// TwinCAT 3 PLC project TcSparkplug
// Title: TcSparkplug
// Company: bstiffler582
// ProjectVersion: 0.0.1
// ProgramVersion: 3.1.4026.22
// libraries:
//   Tc2_Utilities, * (Beckhoff Automation GmbH)
//   Tc2_Standard, * (Beckhoff Automation GmbH)
//   Tc2_System, * (Beckhoff Automation GmbH)
//   Tc3_IotBase, * (Beckhoff Automation GmbH)
// project tree:
//   Util/ F_GetUnixTimestampMs.TcPOU
//   Proto/Enums/ E_ProtoWireType.TcDUT
//   Proto/ FB_ProtoReader.TcPOU, FB_ProtoWriter.TcPOU
//   Sparkplug/Enums/ E_SparkplugState.TcDUT, E_SparkplugDataType.TcDUT, E_SparkplugMessageType.TcDUT
//   Sparkplug/ F_BuildSparkplugTopic.TcPOU, FB_DDeathBuilder.TcPOU, FB_NBirthBuilder.TcPOU, FB_NDeathBuilder.TcPOU, FB_SparkplugPayload.TcPOU, FB_SparkplugDevice.TcPOU, I_SparkplugSession.TcPOU, I_SparkplugDevice.TcPOU, ST_MetricDescriptor.TcDUT, FB_SparkplugSession.TcPOU
//   Tests/ F_Assert.TcPOU, PRG_ProtoTests.TcPOU, PRG_SparkplugPayloadTests.TcPOU
// (motion and I/O tree: see PLC project test)
// real-time tasks:
//   TASK PlcTask: cycle T#10ms, priority 20, ADS port 350
//   TASK PlcTask1: cycle T#10ms, priority 21, ADS port 351

// ---- Proto/Enums/E_ProtoWireType.TcDUT
{attribute 'qualified_only'}
{attribute 'to_string'}
TYPE E_ProtoWireType :
(
	Varint          := 0,
	Fixed64         := 1,
	LengthDelimited := 2,
	Fixed32         := 5
);
END_TYPE

// ---- Sparkplug/Enums/E_SparkplugState.TcDUT
{attribute 'qualified_only'}
{attribute 'to_string'}
TYPE E_SparkplugState :
(
	Idle         := 0,	// Not started or cleanly stopped
	Connecting   := 1,	// MQTT connect in progress
	Birthing     := 2,	// NBIRTH published; waiting one cycle for device DBIRTHs
	Online       := 3,	// Fully operational
	Reconnecting := 4	// Connection lost; waiting before retry
);
END_TYPE

// ---- Sparkplug/Enums/E_SparkplugDataType.TcDUT
{attribute 'qualified_only'}
{attribute 'to_string'}
// Sparkplug B data type codes as defined in the specification.
// These are written into the `datatype` field (field 4) of every Metric.
TYPE E_SparkplugDataType :
(
	Unknown  := 0,
	Int8     := 1,
	Int16    := 2,
	Int32    := 3,
	Int64    := 4,
	UInt8    := 5,
	UInt16   := 6,
	UInt32   := 7,
	UInt64   := 8,
	Float    := 9,
	Double   := 10,
	Boolean  := 11,
	String_   := 12,
	DateTime := 13,
	Text     := 14,
	UUID     := 15,
	DataSet  := 16,
	Bytes    := 17,
	File_    := 18,   // 'File' is a reserved word in some TwinCAT versions
	Template := 19
);
END_TYPE

// ---- Sparkplug/Enums/E_SparkplugMessageType.TcDUT
{attribute 'qualified_only'}
{attribute 'to_string'}
// Sparkplug B message types.
// Note: STATE topics use a different structure (spBv1.0/STATE/{scada_host_id})
// and are handled separately in the session manager.
TYPE E_SparkplugMessageType :
(
	NBIRTH := 0,
	NDEATH := 1,
	DBIRTH := 2,
	DDEATH := 3,
	NDATA  := 4,
	DDATA  := 5,
	NCMD   := 6,
	DCMD   := 7
);
END_TYPE

// ---- Sparkplug/ST_MetricDescriptor.TcDUT
// Describes a single metric registered via FB_SparkplugDevice.AddMetric.
//
// pValue is a live pointer to the original variable in the caller's scope —
// it is dereferenced on every encode, so metric values are always current.
//
// aLastValue / sLastString hold the last-published value for change detection.
// They are updated by FB_SparkplugDevice._syncShadows() after each successful publish.
// fDeadband applies to REAL and LREAL metrics only; 0.0 means any change triggers a publish.
TYPE ST_MetricDescriptor :
STRUCT
	sName		: STRING(255);				// metric name (written in BIRTH messages)
	nAlias		: ULINT;					// alias (written in BIRTH; used alone in DATA)
	eDataType	: E_SparkplugDataType;		// Sparkplug B type code written in the metric header
	eTypeClass	: __SYSTEM.TYPE_CLASS;		// IEC type class — determines how pValue is dereferenced
	pValue		: PVOID;					// pointer to the live variable in the caller's scope
	// Change detection shadow — updated on every successful publish
	aLastValue	: ARRAY[0..7] OF BYTE;		// last-published value for non-string types (max 8 bytes)
	sLastString	: STRING(255);				// last-published value for STRING metrics
	fDeadband	: LREAL;					// minimum change to trigger a publish (REAL/LREAL only)
	bChanged	: BOOL;						// TRUE when live value differs from last-published shadow
END_STRUCT
END_TYPE

// ---- Sparkplug/I_SparkplugSession.TcPOU
// Interface consumed by device FBs to interact with the Sparkplug session.
// Decouples device FBs from the concrete FB_SparkplugSession type,
// enabling testability without a live MQTT connection.
INTERFACE I_SparkplugSession

// Returns the current seq counter and advances it (0–255 wrapping).
// Call once per outbound message to stamp the payload header.
METHOD GetNextSeq : ULINT
END_METHOD

// Returns TRUE when the session is in the Online state.
METHOD IsOnline : BOOL
END_METHOD

// Publishes a pre-encoded payload to the broker.
// Only succeeds when the session is Online or Birthing.
METHOD Publish : BOOL
VAR_INPUT
	sTopic		: STRING(255);
	pPayload	: POINTER TO BYTE;
	nLen		: UDINT;
	nQos		: UDINT;
	bRetain		: BOOL;
END_VAR
END_METHOD

// Sparkplug group ID — used by device FBs to build their own topics.
PROPERTY GroupId : STRING(127)
GET
END_GET
END_PROPERTY

// Sparkplug node ID — used by device FBs to build their own topics.
PROPERTY NodeId : STRING(127)
GET
END_GET
END_PROPERTY

END_INTERFACE

// ---- Sparkplug/I_SparkplugDevice.TcPOU
// Interface implemented by device FBs and consumed by FB_SparkplugSession
// to orchestrate the birth cycle and device lifecycle.
INTERFACE I_SparkplugDevice

// Called by the session at the start of each birth cycle, after NBIRTH is sent.
// The device must encode and publish its DBIRTH using the session's
// GetNextSeq() and Publish() methods.
METHOD OnBirth
END_METHOD

// Encodes and publishes a DDATA message using the current metric values.
// Returns FALSE if the session is not online or the publish fails.
METHOD PublishData : BOOL
VAR_INPUT
	bChangedOnly		: BOOL  := FALSE;
END_VAR
END_METHOD

// Publishes a DDEATH for this device, signalling the host that it is offline.
// Returns FALSE if the session is not online or the publish fails.
METHOD PublishDeath : BOOL
END_METHOD

// Called by the session when the device is registered via AddDevice.
// The device stores the session reference and device ID for use in OnBirth/PublishData.
METHOD SetSession
VAR_INPUT
	sDeviceId	: STRING(127);
	ipSession	: I_SparkplugSession;
END_VAR
END_METHOD

END_INTERFACE

// ---- Util/F_GetUnixTimestampMs.TcPOU
// Returns the current UTC time as milliseconds since the Unix epoch (1970-01-01 00:00:00 UTC).
// Requires: Tc2_Utilities (for F_GetSystemTime).
// F_GetSystemTime returns a ULINT of 100-nanosecond ticks since 1601-01-01 00:00:00 UTC.
FUNCTION F_GetUnixTimestampMs : ULINT

// 116444736000000000 = number of 100ns ticks from 1601-01-01 to 1970-01-01
//   = 134774 days * 86400 s/day * 10,000,000 ticks/s
// Divide by 10,000 to convert remaining 100ns ticks to milliseconds.
F_GetUnixTimestampMs := (F_GetSystemTime() - 116444736000000000) / 10000;

END_FUNCTION

// ---- Proto/FB_ProtoReader.TcPOU
FUNCTION_BLOCK FB_ProtoReader
VAR_INPUT
END_VAR
VAR_OUTPUT
END_VAR
VAR
	_pBuffer      	: POINTER TO BYTE;
	_nLength      	: UDINT;
	_nPos         	: UDINT;
	_nFieldNumber 	: UDINT;
	_eWireType    	: E_ProtoWireType;
	_bError       	: BOOL;
END_VAR

PROPERTY FieldNumber : UDINT
GET
FieldNumber := _nFieldNumber;
END_GET
END_PROPERTY

PROPERTY HasError : BOOL
GET
HasError := _bError;
END_GET
END_PROPERTY

METHOD Init
VAR_INPUT
	pBuffer 	: POINTER TO BYTE;
	nLength 	: UDINT;
END_VAR
_pBuffer      := pBuffer;
_nLength      := nLength;
_nPos         := 0;
_nFieldNumber := 0;
_bError       := FALSE;
END_METHOD

METHOD Next : BOOL
VAR_INPUT
END_VAR
VAR
	nTag : ULINT;
END_VAR
IF _bError OR _nPos >= _nLength THEN
	Next := FALSE;
	RETURN;
END_IF
IF NOT readVarintRaw(nValue => nTag) THEN
	Next := FALSE;
	RETURN;
END_IF
_nFieldNumber := ULINT_TO_UDINT(SHR(nTag, 3));
_eWireType    := ULINT_TO_INT(nTag AND 16#07);
Next := TRUE;
END_METHOD

METHOD PUBLIC ReadBool : BOOL
VAR_INPUT
END_VAR
VAR_OUTPUT
	bValue 		: BOOL;
END_VAR
VAR
	nRaw		: ULINT;
END_VAR
IF _eWireType <> E_ProtoWireType.Varint THEN _bError := TRUE; RETURN; END_IF
IF readVarintRaw(nValue => nRaw) THEN
	bValue  := nRaw <> 0;
	ReadBool := TRUE;
END_IF
END_METHOD

METHOD PUBLIC ReadBytes : BOOL
VAR_INPUT
END_VAR
VAR_OUTPUT
	pData 		: POINTER TO BYTE;
	nLen  		: UDINT;
END_VAR
VAR
	nLenRaw : ULINT;
END_VAR
IF _eWireType <> E_ProtoWireType.LengthDelimited THEN _bError := TRUE; RETURN; END_IF
IF NOT readVarintRaw(nValue => nLenRaw) THEN RETURN; END_IF
nLen := ULINT_TO_UDINT(nLenRaw);
IF _nPos + nLen > _nLength THEN _bError := TRUE; RETURN; END_IF
pData     := _pBuffer + _nPos;
_nPos     := _nPos + nLen;
ReadBytes := TRUE;
END_METHOD

METHOD PUBLIC ReadDouble : BOOL
VAR_INPUT
END_VAR
VAR_OUTPUT
	fValue 		: LREAL;
END_VAR
IF _eWireType <> E_ProtoWireType.Fixed64 OR _nPos + 8 > _nLength THEN
	_bError := TRUE; RETURN;
END_IF
MEMCPY(destAddr := ADR(fValue), srcAddr := _pBuffer + _nPos, n := 8);
_nPos      := _nPos + 8;
ReadDouble := TRUE;
END_METHOD

METHOD PUBLIC ReadFloat : BOOL
VAR_INPUT
END_VAR
VAR_OUTPUT
	fValue 		: REAL;
END_VAR
IF _eWireType <> E_ProtoWireType.Fixed32 OR _nPos + 4 > _nLength THEN
	_bError := TRUE; RETURN;
END_IF
MEMCPY(destAddr := ADR(fValue), srcAddr := _pBuffer + _nPos, n := 4);
_nPos     := _nPos + 4;
ReadFloat := TRUE;
END_METHOD

METHOD PUBLIC ReadUInt32 : BOOL
VAR_INPUT
END_VAR
VAR_OUTPUT
	nValue 		: UDINT;
END_VAR
VAR
	nRaw		: ULINT;
END_VAR
IF _eWireType <> E_ProtoWireType.Varint THEN _bError := TRUE; RETURN; END_IF
IF readVarintRaw(nValue => nRaw) THEN
	nValue    	:= ULINT_TO_UDINT(nRaw);
	ReadUInt32 	:= TRUE;
END_IF
END_METHOD

METHOD PUBLIC ReadUInt64 : BOOL
VAR_INPUT
END_VAR
VAR_OUTPUT
	nValue 		: ULINT;
END_VAR
IF _eWireType <> E_ProtoWireType.Varint THEN _bError := TRUE; RETURN; END_IF
ReadUInt64 := readVarintRaw(nValue => nValue);
END_METHOD

METHOD PRIVATE readVarintRaw : BOOL
VAR_INPUT
END_VAR
VAR_OUTPUT
	nValue 		: ULINT;
END_VAR
VAR
	nByte  		: BYTE;
	nShift 		: BYTE := 0;
END_VAR
nValue := 0;
REPEAT
	IF _nPos >= _nLength THEN
		_bError := TRUE;
		readVarintRaw := FALSE;
		RETURN;
	END_IF
	nByte  := _pBuffer[_nPos];
	_nPos  := _nPos + 1;
	nValue := nValue OR SHL(BYTE_TO_ULINT(nByte AND 16#7F), nShift);
	nShift := nShift + 7;
UNTIL (nByte AND 16#80) = 0 OR nShift >= 64
END_REPEAT;
readVarintRaw := TRUE;
END_METHOD

METHOD Skip : BOOL
VAR_INPUT
END_VAR
VAR
	nLen 		: ULINT;
END_VAR
CASE _eWireType OF
	E_ProtoWireType.Varint:
		Skip := readVarintRaw(nValue=>);  // discard
	E_ProtoWireType.Fixed32:
		IF _nPos + 4 <= _nLength THEN _nPos := _nPos + 4; Skip := TRUE; END_IF
	E_ProtoWireType.Fixed64:
		IF _nPos + 8 <= _nLength THEN _nPos := _nPos + 8; Skip := TRUE; END_IF
	E_ProtoWireType.LengthDelimited:
		IF readVarintRaw(nValue => nLen) THEN
			_nPos := _nPos + ULINT_TO_UDINT(nLen);
			Skip  := _nPos <= _nLength;
		END_IF
	ELSE
		_bError := TRUE;
END_CASE
END_METHOD

METHOD PUBLIC ReadString : BOOL
VAR_INPUT
END_VAR
VAR_OUTPUT
	sValue	: STRING(255);
END_VAR
VAR
	pData	: POINTER TO BYTE;
	nLen	: UDINT;
	nCopy	: UDINT;
	pNull	: POINTER TO BYTE;
END_VAR
IF NOT ReadBytes(pData => pData, nLen => nLen) THEN RETURN; END_IF
nCopy := MIN(nLen, 255);
MEMCPY(destAddr := ADR(sValue), srcAddr := pData, n := nCopy);
// Write null terminator at the end of the copied content
pNull  := ADR(sValue) + nCopy;
pNull^ := 0;
ReadString := TRUE;
END_METHOD

PROPERTY WireType : E_ProtoWireType
GET
WireType := _eWireType;
END_GET
END_PROPERTY

END_FUNCTION_BLOCK

// ---- Proto/FB_ProtoWriter.TcPOU
FUNCTION_BLOCK FB_ProtoWriter
VAR_INPUT
END_VAR
VAR_OUTPUT
END_VAR
VAR
	_pBuffer    	: POINTER TO BYTE;
	_nCapacity  	: UDINT;
	_nLength    	: UDINT;
	_bError     	: BOOL;
END_VAR

// Pointer to the start of the encoded bytes. Valid until the next Init call.
PROPERTY Buffer : POINTER TO BYTE
GET
Buffer := _pBuffer;
END_GET
END_PROPERTY

PROPERTY HasError : BOOL
GET
HasError := _bError;
END_GET
END_PROPERTY

METHOD Init
VAR_INPUT
	pBuffer		 		: POINTER TO BYTE;
	nCapacity			: UDINT;
END_VAR
_pBuffer   := pBuffer;
_nCapacity := nCapacity;
_nLength   := 0;
_bError    := FALSE;
END_METHOD

PROPERTY Length : UDINT
GET
Length := _nLength;
END_GET
END_PROPERTY

METHOD Reset : PVOID
VAR_INPUT
END_VAR
_nLength := 0;
_bError  := FALSE;
END_METHOD

METHOD PUBLIC WriteBool : BOOL
VAR_INPUT
	nFieldNumber 	: UDINT;
	bValue       	: BOOL;
END_VAR
WriteBool := writeTag(nFieldNumber, E_ProtoWireType.Varint)
	AND writeVarint(BOOL_TO_ULINT(bValue));
END_METHOD

METHOD PUBLIC WriteBytes : BOOL
VAR_INPUT
	nFieldNumber 	: UDINT;
	pData        	: POINTER TO BYTE;
	nLen         	: UDINT;
END_VAR
WriteBytes := writeTag(nFieldNumber, E_ProtoWireType.LengthDelimited)
	AND writeVarint(UDINT_TO_ULINT(nLen))
	AND writeRawBytes(pData, nLen);
END_METHOD

METHOD PUBLIC WriteDouble : BOOL
VAR_INPUT
	nFieldNumber 	: UDINT;
	fValue       	: LREAL;
END_VAR
VAR
	nRaw			: LWORD;
END_VAR
MEMCPY(destAddr := ADR(nRaw), srcAddr := ADR(fValue), n := 8);
WriteDouble := writeTag(nFieldNumber, E_ProtoWireType.Fixed64)
	AND writeRawBytes(ADR(nRaw), 8);
END_METHOD

METHOD PUBLIC WriteFloat : BOOL
VAR_INPUT
	nFieldNumber 	: UDINT;
	fValue       	: REAL;
END_VAR
VAR
	nRaw			: DWORD;
END_VAR
MEMCPY(destAddr := ADR(nRaw), srcAddr := ADR(fValue), n := 4);
WriteFloat := writeTag(nFieldNumber, E_ProtoWireType.Fixed32)
	AND writeRawBytes(ADR(nRaw), 4);
END_METHOD

METHOD PRIVATE writeRawByte : BOOL
VAR_INPUT
	nByte		: BYTE;
END_VAR
IF _bError OR _nLength >= _nCapacity THEN
	_bError := TRUE;
	writeRawByte := FALSE;
	RETURN;
END_IF
_pBuffer[_nLength] := nByte;
_nLength := _nLength + 1;
writeRawByte := TRUE;
END_METHOD

METHOD PRIVATE writeRawBytes : BOOL
VAR_INPUT
	pData : POINTER TO BYTE;
	nLen  : UDINT;
END_VAR
IF _bError OR (_nLength + nLen > _nCapacity) THEN
	_bError := TRUE;
	writeRawBytes := FALSE;
	RETURN;
END_IF
MEMCPY(destAddr := _pBuffer + _nLength, srcAddr := pData, n := nLen);
_nLength := _nLength + nLen;
writeRawBytes := TRUE;
END_METHOD

METHOD PUBLIC WriteString : BOOL
VAR_INPUT
	nFieldNumber 	: UDINT;
	sValue       	: STRING(255);
END_VAR
VAR
	nLen			: INT;
END_VAR
nLen := LEN(sValue);
WriteString := writeTag(nFieldNumber, E_ProtoWireType.LengthDelimited)
	AND writeVarint(TO_ULINT(nLen))
	AND writeRawBytes(ADR(sValue), TO_UDINT(nLen));
END_METHOD

METHOD PRIVATE writeTag : BOOL
VAR_INPUT
	nFieldNumber 	: UDINT;
	eWireType    	: E_ProtoWireType;
END_VAR
writeTag := writeVarint(
	SHL(UDINT_TO_ULINT(nFieldNumber), 3) OR INT_TO_ULINT(TO_INT(eWireType))
);
END_METHOD

METHOD PUBLIC WriteUInt32 : BOOL
VAR_INPUT
	nFieldNumber 	: UDINT;
	nValue       	: UDINT;
END_VAR
WriteUInt32 := writeTag(nFieldNumber, E_ProtoWireType.Varint)
	AND writeVarint(UDINT_TO_ULINT(nValue));
END_METHOD

METHOD PUBLIC WriteUInt64 : BOOL
VAR_INPUT
	nFieldNumber 	: UDINT;
  	nValue       	: ULINT;
END_VAR
WriteUInt64 := writeTag(nFieldNumber, E_ProtoWireType.Varint)
	AND writeVarint(nValue);
END_METHOD

METHOD PRIVATE writeVarint : BOOL
VAR_INPUT
	nValue		: ULINT;
END_VAR
VAR
	nByte		: BYTE;
END_VAR
IF _bError THEN writeVarint := FALSE; RETURN; END_IF
REPEAT
	nByte  := ULINT_TO_BYTE(nValue AND 16#7F);
	nValue := SHR(nValue, 7);
	IF nValue <> 0 THEN
  		nByte := nByte OR 16#80;  // more bytes follow
	END_IF
	IF NOT writeRawByte(nByte) THEN
		writeVarint := FALSE;
		RETURN;
	END_IF
UNTIL nValue = 0
END_REPEAT;
writeVarint := TRUE;
END_METHOD

END_FUNCTION_BLOCK

// ---- Sparkplug/F_BuildSparkplugTopic.TcPOU
// Builds a Sparkplug B topic string.
//
// Node-level:   spBv1.0/{group_id}/{msg_type}/{node_id}
// Device-level: spBv1.0/{group_id}/{msg_type}/{node_id}/{device_id}
//
// Pass sDeviceId := '' for node-level messages (NBIRTH, NDEATH, NDATA, NCMD).
FUNCTION F_BuildSparkplugTopic : STRING(255)
VAR_INPUT
	eMsgType	: E_SparkplugMessageType;
	sGroupId	: STRING(127);
	sNodeId		: STRING(127);
	sDeviceId	: STRING(127);
END_VAR
VAR
	sMsgType	: STRING(16);
END_VAR

CASE eMsgType OF
	E_SparkplugMessageType.NBIRTH:	sMsgType := 'NBIRTH';
	E_SparkplugMessageType.NDEATH:	sMsgType := 'NDEATH';
	E_SparkplugMessageType.DBIRTH:	sMsgType := 'DBIRTH';
	E_SparkplugMessageType.DDEATH:	sMsgType := 'DDEATH';
	E_SparkplugMessageType.NDATA:	sMsgType := 'NDATA';
	E_SparkplugMessageType.DDATA:	sMsgType := 'DDATA';
	E_SparkplugMessageType.NCMD:	sMsgType := 'NCMD';
	E_SparkplugMessageType.DCMD:	sMsgType := 'DCMD';
	ELSE							sMsgType := 'UNKNOWN';
END_CASE

F_BuildSparkplugTopic := CONCAT('spBv1.0/', sGroupId);
F_BuildSparkplugTopic := CONCAT(F_BuildSparkplugTopic, CONCAT('/', sMsgType));
F_BuildSparkplugTopic := CONCAT(F_BuildSparkplugTopic, CONCAT('/', sNodeId));

IF LEN(sDeviceId) > 0 THEN
	F_BuildSparkplugTopic := CONCAT(F_BuildSparkplugTopic, CONCAT('/', sDeviceId));
END_IF

END_FUNCTION

// ---- Sparkplug/FB_DDeathBuilder.TcPOU
// Builds a Sparkplug B DDEATH payload.
//
// DDEATH announces that a logical device is going offline. It carries only a
// timestamp and seq — no metrics. The session manager publishes it before
// disconnecting a device or on detecting a device fault.
FUNCTION_BLOCK FB_DDeathBuilder
VAR
	_aBuf		: ARRAY[0..31] OF BYTE;
	_fbPayload	: FB_SparkplugPayload;
END_VAR

// FB body intentionally empty — all logic is in Build().

METHOD Build : BOOL
VAR_INPUT
	nTimestamp	: ULINT;
	nSeq		: ULINT;
END_VAR
_fbPayload.Init(ADR(_aBuf), SIZEOF(_aBuf));
_fbPayload.WriteHeader(nTimestamp, nSeq);
Build := NOT _fbPayload.HasError;
END_METHOD

PROPERTY Payload : REFERENCE TO FB_SparkplugPayload
GET
Payload REF= _fbPayload;
END_GET
END_PROPERTY

END_FUNCTION_BLOCK

// ---- Sparkplug/FB_SparkplugPayload.TcPOU
// Incremental Sparkplug B payload builder.
//
// Wraps FB_ProtoWriter with Sparkplug-aware metric write methods. The caller
// provides an external buffer so payload capacity can be sized appropriately
// for the message type (large for NBIRTH/DBIRTH, small for DDATA).
//
// Usage:
//   fbPayload.Init(pBuffer, nCapacity);
//   fbPayload.WriteHeader(nTimestamp, nSeq);
//   fbPayload.WriteBoolMetric('MotorRunning', 1, E_SparkplugDataType.Boolean, TRUE);
//   fbPayload.WriteUInt32Metric('', 2, E_SparkplugDataType.UInt32, nSpeed);  // DATA mode: no name
//   // publish fbPayload.Buffer for fbPayload.Length bytes
//
// Metric name conventions:
//   BIRTH messages  — pass the metric name; alias is also included for future DATA messages.
//   DATA messages   — pass sName := '' to omit the name and use alias only (saves bandwidth).
//   System metrics  — pass nAlias := 0 to omit the alias field (name-only, e.g. bdSeq).
FUNCTION_BLOCK FB_SparkplugPayload
VAR
	_fbPayload		: FB_ProtoWriter;				// outer Payload message
	_fbMetric		: FB_ProtoWriter;				// inner Metric message (reused per metric)
	_aBufMetric		: ARRAY[0..511] OF BYTE;		// temp buffer for one encoded Metric
END_VAR

// FB body intentionally empty — all logic is in the methods below.

// Binds the payload builder to an external buffer and resets it.
// Must be called before any Write methods.
METHOD Init
VAR_INPUT
	pBuffer		: POINTER TO BYTE;
	nCapacity	: UDINT;
END_VAR
_fbPayload.Init(pBuffer, nCapacity);
END_METHOD

// Resets the write position without re-binding the buffer.
// Use when re-encoding into the same buffer (e.g. periodic DDATA).
METHOD Reset
_fbPayload.Reset();
END_METHOD

// Writes the Payload-level timestamp (field 1) and seq (field 4).
// Must be the first Write call after Init/Reset.
//
// Sparkplug field numbers for Payload (from sparkplug_b.proto):
//   1 = timestamp (uint64, ms since Unix epoch)
//   2 = metrics   (repeated, length-delimited)
//   3 = seq       (uint64, 0–255 wrapping)
//   4 = uuid      (string — not used by this library)
METHOD WriteHeader : BOOL
VAR_INPUT
	nTimestamp	: ULINT;
	nSeq		: ULINT;
END_VAR
WriteHeader := _fbPayload.WriteUInt64(1, nTimestamp)
	AND _fbPayload.WriteUInt64(3, nSeq);
END_METHOD

METHOD WriteBoolMetric : BOOL
VAR_INPUT
	sName		: STRING(255);
	nAlias		: ULINT;
	eDataType	: E_SparkplugDataType;
	bValue		: BOOL;
END_VAR
_fbMetric.Init(ADR(_aBufMetric), SIZEOF(_aBufMetric));
IF LEN(sName) > 0  THEN _fbMetric.WriteString(1, sName); END_IF
IF nAlias > 0      THEN _fbMetric.WriteUInt64(2, nAlias); END_IF
_fbMetric.WriteUInt32(4, TO_UDINT(eDataType));
_fbMetric.WriteBool(14, bValue);
WriteBoolMetric := _fbPayload.WriteBytes(2, ADR(_aBufMetric), _fbMetric.Length);
END_METHOD

// For Int8, Int16, Int32, UInt8, UInt16, UInt32 — encoded in proto field 10 (int_value).
METHOD WriteUInt32Metric : BOOL
VAR_INPUT
	sName		: STRING(255);
	nAlias		: ULINT;
	eDataType	: E_SparkplugDataType;
	nValue		: UDINT;
END_VAR
_fbMetric.Init(ADR(_aBufMetric), SIZEOF(_aBufMetric));
IF LEN(sName) > 0  THEN _fbMetric.WriteString(1, sName); END_IF
IF nAlias > 0      THEN _fbMetric.WriteUInt64(2, nAlias); END_IF
_fbMetric.WriteUInt32(4, TO_UDINT(eDataType));
_fbMetric.WriteUInt32(10, nValue);
WriteUInt32Metric := _fbPayload.WriteBytes(2, ADR(_aBufMetric), _fbMetric.Length);
END_METHOD

// For Int64, UInt64, DateTime — encoded in proto field 11 (long_value).
METHOD WriteUInt64Metric : BOOL
VAR_INPUT
	sName		: STRING(255);
	nAlias		: ULINT;
	eDataType	: E_SparkplugDataType;
	nValue		: ULINT;
END_VAR
_fbMetric.Init(ADR(_aBufMetric), SIZEOF(_aBufMetric));
IF LEN(sName) > 0  THEN _fbMetric.WriteString(1, sName); END_IF
IF nAlias > 0      THEN _fbMetric.WriteUInt64(2, nAlias); END_IF
_fbMetric.WriteUInt32(4, TO_UDINT(eDataType));
_fbMetric.WriteUInt64(11, nValue);
WriteUInt64Metric := _fbPayload.WriteBytes(2, ADR(_aBufMetric), _fbMetric.Length);
END_METHOD

METHOD WriteFloatMetric : BOOL
VAR_INPUT
	sName		: STRING(255);
	nAlias		: ULINT;
	eDataType	: E_SparkplugDataType;
	fValue		: REAL;
END_VAR
_fbMetric.Init(ADR(_aBufMetric), SIZEOF(_aBufMetric));
IF LEN(sName) > 0  THEN _fbMetric.WriteString(1, sName); END_IF
IF nAlias > 0      THEN _fbMetric.WriteUInt64(2, nAlias); END_IF
_fbMetric.WriteUInt32(4, TO_UDINT(eDataType));
_fbMetric.WriteFloat(12, fValue);
WriteFloatMetric := _fbPayload.WriteBytes(2, ADR(_aBufMetric), _fbMetric.Length);
END_METHOD

METHOD WriteDoubleMetric : BOOL
VAR_INPUT
	sName		: STRING(255);
	nAlias		: ULINT;
	eDataType	: E_SparkplugDataType;
	fValue		: LREAL;
END_VAR
_fbMetric.Init(ADR(_aBufMetric), SIZEOF(_aBufMetric));
IF LEN(sName) > 0  THEN _fbMetric.WriteString(1, sName); END_IF
IF nAlias > 0      THEN _fbMetric.WriteUInt64(2, nAlias); END_IF
_fbMetric.WriteUInt32(4, TO_UDINT(eDataType));
_fbMetric.WriteDouble(13, fValue);
WriteDoubleMetric := _fbPayload.WriteBytes(2, ADR(_aBufMetric), _fbMetric.Length);
END_METHOD

// For String, Text, UUID data types.
METHOD WriteStringMetric : BOOL
VAR_INPUT
	sName		: STRING(255);
	nAlias		: ULINT;
	eDataType	: E_SparkplugDataType;
	sValue		: STRING(255);
END_VAR
_fbMetric.Init(ADR(_aBufMetric), SIZEOF(_aBufMetric));
IF LEN(sName) > 0  THEN _fbMetric.WriteString(1, sName); END_IF
IF nAlias > 0      THEN _fbMetric.WriteUInt64(2, nAlias); END_IF
_fbMetric.WriteUInt32(4, TO_UDINT(eDataType));
_fbMetric.WriteString(15, sValue);
WriteStringMetric := _fbPayload.WriteBytes(2, ADR(_aBufMetric), _fbMetric.Length);
END_METHOD

// Pointer to the start of the encoded payload. Valid until the next Init call.
PROPERTY Buffer : POINTER TO BYTE
GET
Buffer := _fbPayload.Buffer;
END_GET
END_PROPERTY

PROPERTY Length : UDINT
GET
Length := _fbPayload.Length;
END_GET
END_PROPERTY

PROPERTY HasError : BOOL
GET
HasError := _fbPayload.HasError;
END_GET
END_PROPERTY

END_FUNCTION_BLOCK

// ---- Sparkplug/FB_NBirthBuilder.TcPOU
// Builds the Sparkplug B NBIRTH payload.
//
// NBIRTH announces the edge node to the Sparkplug host. It must be published
// immediately after the MQTT connection is established, before any DBIRTH or
// data messages. The seq counter is reset to 0 on every NBIRTH.
//
// This builder writes the two mandatory Sparkplug system metrics:
//   "bdSeq"                — UInt64, the birth/death sequence number.
//   "Node Control/Rebirth" — Boolean, always FALSE in the birth payload.
//                            The host writes TRUE to this metric (via NCMD)
//                            to request a full rebirth cycle.
//
// Generated code calls Payload to append node-level user metrics after Build().
//
// Usage (session manager):
//   fbNBirth.Build(nTimestamp, nBdSeq);
//   // generated node-level metrics (if any):
//   fbNBirth.Payload.WriteBoolMetric('MyNodeMetric', 1, Boolean, bValue);
//   mqttClient.Publish(sTopic, fbNBirth.Payload.Buffer, fbNBirth.Payload.Length);
FUNCTION_BLOCK FB_NBirthBuilder
VAR
	_aBuf		: ARRAY[0..2047] OF BYTE;	// 2 KB — generous for node metrics
	_fbPayload	: FB_SparkplugPayload;
END_VAR

// FB body intentionally empty — all logic is in Build().

// Initialises the payload and writes the header + system metrics.
// Call this once after connecting, before publishing NBIRTH.
// After this call, append any node-level user metrics via the Payload property.
METHOD Build : BOOL
VAR_INPUT
	nTimestamp	: ULINT;	// ms since Unix epoch
	nBdSeq		: ULINT;	// birth/death sequence number (0–255 wrapping, RETAIN)
END_VAR
_fbPayload.Init(ADR(_aBuf), SIZEOF(_aBuf));

// seq is always 0 for NBIRTH — the counter resets on every birth.
_fbPayload.WriteHeader(nTimestamp, 0);

// bdSeq: no alias — the host identifies this metric by name.
_fbPayload.WriteUInt64Metric('bdSeq', 0, E_SparkplugDataType.UInt64, nBdSeq);

// Node Control/Rebirth: no alias — identified by name.
// Value is always FALSE in the birth payload; the host sends TRUE via NCMD
// to trigger a rebirth.
_fbPayload.WriteBoolMetric('Node Control/Rebirth', 0, E_SparkplugDataType.Boolean, FALSE);

Build := NOT _fbPayload.HasError;
END_METHOD

// Exposes the underlying payload builder so generated code can append
// node-level user metrics after Build() is called.
PROPERTY Payload : REFERENCE TO FB_SparkplugPayload
GET
Payload REF= _fbPayload;
END_GET
END_PROPERTY

END_FUNCTION_BLOCK

// ---- Sparkplug/FB_NDeathBuilder.TcPOU
// Builds a Sparkplug B NDEATH payload.
//
// NDEATH is the MQTT Will message — it must be pre-built and registered with the
// broker before the MQTT connection is established. When the broker detects an
// ungraceful disconnect it publishes this payload automatically.
//
// The NDEATH payload contains exactly one metric:
//   Metric { name: "bdSeq", datatype: UInt64, long_value: <bdSeq> }
//
// No timestamp and no seq field are included per the Sparkplug B specification.
//
// Usage:
//   fbNDeath.Build(nBdSeq);
//   mqttClient.SetWill(
//     sTopic  := F_BuildSparkplugTopic(NDEATH, sGroup, sNode, ''),
//     pPayload := fbNDeath.PayloadBuffer,
//     nLen     := fbNDeath.PayloadLength);
FUNCTION_BLOCK FB_NDeathBuilder
VAR
	// Internal buffers — owned by this FB, stable between Build() calls.
	_aBufMetric		: ARRAY[0..31] OF BYTE;
	_aBufPayload	: ARRAY[0..47] OF BYTE;

	_fbMetric		: FB_ProtoWriter;
	_fbPayload		: FB_ProtoWriter;

	_nPayloadLength	: UDINT;
	_bValid			: BOOL;
END_VAR

// FB body intentionally empty — all logic is in Build().

// Encodes the NDEATH payload for the given birth/death sequence number.
// Call this once before registering the MQTT Will, and again after each
// reconnect if the bdSeq value has changed.
METHOD Build : BOOL
VAR_INPUT
	nBdSeq	: ULINT;
END_VAR
// ── Encode the bdSeq metric ──────────────────────────────────────────────────
// Sparkplug field numbers for Metric:
//   1 = name (string)
//   4 = datatype (uint32)
//  11 = long_value (uint64) — used for UInt64 and Int64 values
_fbMetric.Init(ADR(_aBufMetric), SIZEOF(_aBufMetric));
_fbMetric.WriteString(1,  'bdSeq');
_fbMetric.WriteUInt32(4,  TO_UDINT(E_SparkplugDataType.UInt64));
_fbMetric.WriteUInt64(11, nBdSeq);

// ── Encode the Payload ────────────────────────────────────────────────────────
// Sparkplug field numbers for Payload:
//   2 = metrics (repeated, length-delimited)
// Intentionally omitting timestamp (f1) and seq (f4) — not required in NDEATH.
_fbPayload.Init(ADR(_aBufPayload), SIZEOF(_aBufPayload));
_fbPayload.WriteBytes(2, ADR(_aBufMetric), _fbMetric.Length);

_bValid         := NOT _fbMetric.HasError AND NOT _fbPayload.HasError;
_nPayloadLength := _fbPayload.Length;
Build           := _bValid;
END_METHOD

// TRUE if the last Build() call succeeded without buffer overflow.
PROPERTY IsValid : BOOL
GET
IsValid := _bValid;
END_GET
END_PROPERTY

// Pointer to the encoded payload bytes. Valid until the next Build() call.
PROPERTY PayloadBuffer : POINTER TO BYTE
GET
PayloadBuffer := ADR(_aBufPayload);
END_GET
END_PROPERTY

// Number of encoded bytes. Zero if Build() has not been called yet.
PROPERTY PayloadLength : UDINT
GET
PayloadLength := _nPayloadLength;
END_GET
END_PROPERTY

END_FUNCTION_BLOCK

// ---- Sparkplug/FB_SparkplugDevice.TcPOU
// Generic Sparkplug B device function block.
//
// Register metrics once at startup via AddMetric(), then pass this FB to the
// session via AddDevice(). The session will call OnBirth() automatically on
// every birth cycle; the caller decides when to send DDATA by calling PublishData().
//
// Usage:
//   fbDevice.AddMetric('Speed',       1, nMotorSpeed);
//   fbDevice.AddMetric('Running',     2, bMotorRunning);
//   fbDevice.AddMetric('Temperature', 3, fMotorTemp);
//   fbSpkSession.AddDevice('Motor1', fbDevice);
//   // ...
//   IF tPublish.Q THEN fbDevice.PublishData(); END_IF
//
// AddMetric() stores a live pointer to the caller's variable — do not call it
// more than once per metric, and ensure the variable outlives this FB.
//
// Call this FB every PLC cycle. It runs change detection and sets bDataPending
// when at least one metric's live value differs from its last-published shadow.
// The caller then decides when to call PublishData() (e.g. on bDataPending rising edge).
FUNCTION_BLOCK FB_SparkplugDevice IMPLEMENTS I_SparkplugDevice
VAR_INPUT
	// Default deadband applied to all REAL and LREAL metrics at AddMetric time.
	// Per-metric overrides are available via SetDeadband(). 0.0 = any change triggers a publish.
	fDefaultDeadband	: LREAL := 0.0;
	// When TRUE the FB publishes DDATA automatically on any detected change.
	// The caller may still call PublishData() independently (e.g. periodic refresh).
	bAutoPublish		: BOOL  := FALSE;
END_VAR
VAR_OUTPUT
	// TRUE when at least one metric's live value differs from its last-published shadow.
	// Recomputed every cycle — if a value changes and reverts before PublishData() is called,
	// this returns FALSE (correct report-by-exception behaviour).
	bDataPending		: BOOL;
END_VAR
VAR
	_aMetrics		: ARRAY[0..15] OF ST_MetricDescriptor;
	_nMetricCount	: UDINT;

	_sDeviceId		: STRING(127);
	_ipSession		: I_SparkplugSession;

	_sBirthTopic	: STRING(255);
	_sDataTopic		: STRING(255);
	_sDeathTopic	: STRING(255);

	_aBirthBuf		: ARRAY[0..2047] OF BYTE;
	_aDataBuf		: ARRAY[0..511] OF BYTE;
	_fbBirthPayload	: FB_SparkplugPayload;
	_fbDataPayload	: FB_SparkplugPayload;
	_fbDeath		: FB_DDeathBuilder;
END_VAR

// Run change detection every cycle once a session is attached.
IF _ipSession <> 0 THEN
	_checkChanges();
	IF bAutoPublish AND bDataPending THEN
		PublishData(bChangedOnly := TRUE);
	END_IF
END_IF

// Encodes all registered metrics into fbPayload.
// bBirthMode = TRUE  → writes name + alias (DBIRTH).
// bBirthMode = FALSE → writes alias only (DDATA — saves bandwidth).
METHOD PRIVATE _writeMetrics
VAR_IN_OUT
	fbPayload	: FB_SparkplugPayload;
END_VAR
VAR_INPUT
	bBirthMode		: BOOL;
	bChangedOnly	: BOOL := FALSE;	// when TRUE, skips metrics whose bChanged flag is FALSE
END_VAR
VAR
	i		: UDINT;
	sName	: STRING(255);
	pBool	: POINTER TO BOOL;
	pSint	: POINTER TO SINT;
	pInt	: POINTER TO INT;
	pDint	: POINTER TO DINT;
	pLint	: POINTER TO LINT;
	pUsint	: POINTER TO USINT;
	pUint	: POINTER TO UINT;
	pUdint	: POINTER TO UDINT;
	pUlint	: POINTER TO ULINT;
	pByte	: POINTER TO BYTE;
	pWord	: POINTER TO WORD;
	pDword	: POINTER TO DWORD;
	pLword	: POINTER TO LWORD;
	pReal	: POINTER TO REAL;
	pLreal	: POINTER TO LREAL;
	pStr	: POINTER TO STRING(255);
END_VAR
IF _nMetricCount = 0 THEN RETURN; END_IF

FOR i := 0 TO _nMetricCount - 1 DO
	// In changed-only mode skip metrics that haven't changed since last publish.
	IF bChangedOnly AND NOT _aMetrics[i].bChanged THEN
		;
	ELSE
	// In BIRTH mode write the metric name; in DATA mode write alias only.
	sName := SEL(bBirthMode, '', _aMetrics[i].sName);

	CASE _aMetrics[i].eTypeClass OF
		__SYSTEM.TYPE_CLASS.TYPE_BOOL:
			pBool  := _aMetrics[i].pValue;
			fbPayload.WriteBoolMetric(sName, _aMetrics[i].nAlias, _aMetrics[i].eDataType, pBool^);

		__SYSTEM.TYPE_CLASS.TYPE_SINT:
			pSint  := _aMetrics[i].pValue;
			fbPayload.WriteUInt32Metric(sName, _aMetrics[i].nAlias, _aMetrics[i].eDataType, TO_UDINT(pSint^));

		__SYSTEM.TYPE_CLASS.TYPE_INT:
			pInt   := _aMetrics[i].pValue;
			fbPayload.WriteUInt32Metric(sName, _aMetrics[i].nAlias, _aMetrics[i].eDataType, TO_UDINT(pInt^));

		__SYSTEM.TYPE_CLASS.TYPE_DINT:
			pDint  := _aMetrics[i].pValue;
			fbPayload.WriteUInt32Metric(sName, _aMetrics[i].nAlias, _aMetrics[i].eDataType, TO_UDINT(pDint^));

		__SYSTEM.TYPE_CLASS.TYPE_LINT:
			pLint  := _aMetrics[i].pValue;
			fbPayload.WriteUInt64Metric(sName, _aMetrics[i].nAlias, _aMetrics[i].eDataType, TO_ULINT(pLint^));

		__SYSTEM.TYPE_CLASS.TYPE_USINT:
			pUsint := _aMetrics[i].pValue;
			fbPayload.WriteUInt32Metric(sName, _aMetrics[i].nAlias, _aMetrics[i].eDataType, TO_UDINT(pUsint^));

		__SYSTEM.TYPE_CLASS.TYPE_UINT:
			pUint  := _aMetrics[i].pValue;
			fbPayload.WriteUInt32Metric(sName, _aMetrics[i].nAlias, _aMetrics[i].eDataType, TO_UDINT(pUint^));

		__SYSTEM.TYPE_CLASS.TYPE_UDINT:
			pUdint := _aMetrics[i].pValue;
			fbPayload.WriteUInt32Metric(sName, _aMetrics[i].nAlias, _aMetrics[i].eDataType, pUdint^);

		__SYSTEM.TYPE_CLASS.TYPE_ULINT:
			pUlint := _aMetrics[i].pValue;
			fbPayload.WriteUInt64Metric(sName, _aMetrics[i].nAlias, _aMetrics[i].eDataType, pUlint^);

		__SYSTEM.TYPE_CLASS.TYPE_BYTE:
			pByte  := _aMetrics[i].pValue;
			fbPayload.WriteUInt32Metric(sName, _aMetrics[i].nAlias, _aMetrics[i].eDataType, TO_UDINT(pByte^));

		__SYSTEM.TYPE_CLASS.TYPE_WORD:
			pWord  := _aMetrics[i].pValue;
			fbPayload.WriteUInt32Metric(sName, _aMetrics[i].nAlias, _aMetrics[i].eDataType, TO_UDINT(pWord^));

		__SYSTEM.TYPE_CLASS.TYPE_DWORD:
			pDword := _aMetrics[i].pValue;
			fbPayload.WriteUInt32Metric(sName, _aMetrics[i].nAlias, _aMetrics[i].eDataType, TO_UDINT(pDword^));

		__SYSTEM.TYPE_CLASS.TYPE_LWORD:
			pLword := _aMetrics[i].pValue;
			fbPayload.WriteUInt64Metric(sName, _aMetrics[i].nAlias, _aMetrics[i].eDataType, TO_ULINT(pLword^));

		__SYSTEM.TYPE_CLASS.TYPE_REAL:
			pReal  := _aMetrics[i].pValue;
			fbPayload.WriteFloatMetric(sName, _aMetrics[i].nAlias, _aMetrics[i].eDataType, pReal^);

		__SYSTEM.TYPE_CLASS.TYPE_LREAL:
			pLreal := _aMetrics[i].pValue;
			fbPayload.WriteDoubleMetric(sName, _aMetrics[i].nAlias, _aMetrics[i].eDataType, pLreal^);

		__SYSTEM.TYPE_CLASS.TYPE_STRING:
			pStr   := _aMetrics[i].pValue;
			fbPayload.WriteStringMetric(sName, _aMetrics[i].nAlias, _aMetrics[i].eDataType, pStr^);
	END_CASE
	END_IF
END_FOR
END_METHOD

// Registers a metric to be included in DBIRTH and DDATA messages.
// Infers the Sparkplug B data type from the IEC type of value.
// Call once per metric during startup before AddDevice().
//
// Supported types: BOOL, SINT/INT/DINT/LINT, USINT/UINT/UDINT/ULINT,
//                  BYTE/WORD/DWORD/LWORD, REAL, LREAL, STRING(n)
METHOD AddMetric
VAR_INPUT
	sName	: STRING(255);
	nAlias	: ULINT;
	value	: ANY;
END_VAR
VAR
	eDataType	: E_SparkplugDataType;
END_VAR
IF _nMetricCount >= 16 THEN RETURN; END_IF

// Map IEC TypeClass → Sparkplug B data type code
CASE value.TypeClass OF
	__SYSTEM.TYPE_CLASS.TYPE_BOOL	: eDataType := E_SparkplugDataType.Boolean;
	__SYSTEM.TYPE_CLASS.TYPE_SINT	: eDataType := E_SparkplugDataType.Int8;
	__SYSTEM.TYPE_CLASS.TYPE_INT	: eDataType := E_SparkplugDataType.Int16;
	__SYSTEM.TYPE_CLASS.TYPE_DINT	: eDataType := E_SparkplugDataType.Int32;
	__SYSTEM.TYPE_CLASS.TYPE_LINT	: eDataType := E_SparkplugDataType.Int64;
	__SYSTEM.TYPE_CLASS.TYPE_USINT	: eDataType := E_SparkplugDataType.UInt8;
	__SYSTEM.TYPE_CLASS.TYPE_UINT	: eDataType := E_SparkplugDataType.UInt16;
	__SYSTEM.TYPE_CLASS.TYPE_UDINT	: eDataType := E_SparkplugDataType.UInt32;
	__SYSTEM.TYPE_CLASS.TYPE_ULINT	: eDataType := E_SparkplugDataType.UInt64;
	__SYSTEM.TYPE_CLASS.TYPE_BYTE	: eDataType := E_SparkplugDataType.UInt8;
	__SYSTEM.TYPE_CLASS.TYPE_WORD	: eDataType := E_SparkplugDataType.UInt16;
	__SYSTEM.TYPE_CLASS.TYPE_DWORD	: eDataType := E_SparkplugDataType.UInt32;
	__SYSTEM.TYPE_CLASS.TYPE_LWORD	: eDataType := E_SparkplugDataType.UInt64;
	__SYSTEM.TYPE_CLASS.TYPE_REAL	: eDataType := E_SparkplugDataType.Float;
	__SYSTEM.TYPE_CLASS.TYPE_LREAL	: eDataType := E_SparkplugDataType.Double;
	__SYSTEM.TYPE_CLASS.TYPE_STRING	: eDataType := E_SparkplugDataType.String_;
ELSE
	eDataType := E_SparkplugDataType.Unknown;
END_CASE

_aMetrics[_nMetricCount].sName		 := sName;
_aMetrics[_nMetricCount].nAlias		 := nAlias;
_aMetrics[_nMetricCount].eDataType	 := eDataType;
_aMetrics[_nMetricCount].eTypeClass  := value.TypeClass;
_aMetrics[_nMetricCount].pValue		 := value.pValue;

// Apply default deadband to float types; all others use exact-match comparison.
_aMetrics[_nMetricCount].fDeadband := 0.0;
IF value.TypeClass = __SYSTEM.TYPE_CLASS.TYPE_REAL
OR value.TypeClass = __SYSTEM.TYPE_CLASS.TYPE_LREAL THEN
	_aMetrics[_nMetricCount].fDeadband := fDefaultDeadband;
END_IF

_nMetricCount := _nMetricCount + 1;
END_METHOD

// Called by the session on each birth cycle after NBIRTH is published.
// Builds topics, encodes the DBIRTH payload, and publishes it.
METHOD OnBirth
// Build topics — GroupId and NodeId are valid once the session has been called at least once.
_sBirthTopic := F_BuildSparkplugTopic(E_SparkplugMessageType.DBIRTH, _ipSession.GroupId, _ipSession.NodeId, _sDeviceId);
_sDataTopic  := F_BuildSparkplugTopic(E_SparkplugMessageType.DDATA,  _ipSession.GroupId, _ipSession.NodeId, _sDeviceId);
_sDeathTopic := F_BuildSparkplugTopic(E_SparkplugMessageType.DDEATH, _ipSession.GroupId, _ipSession.NodeId, _sDeviceId);

_fbBirthPayload.Init(ADR(_aBirthBuf), SIZEOF(_aBirthBuf));
_fbBirthPayload.WriteHeader(F_GetUnixTimestampMs(), _ipSession.GetNextSeq());
_writeMetrics(_fbBirthPayload, TRUE);
_ipSession.Publish(_sBirthTopic, _fbBirthPayload.Buffer, _fbBirthPayload.Length, 1, FALSE);

// Sync shadows after birth so change detection starts from the just-published values.
_syncShadows();
END_METHOD

// Encodes and publishes a DDATA message.
// bChangedOnly = FALSE (default): sends all metrics — use for periodic refreshes.
// bChangedOnly = TRUE: sends only metrics whose value has changed since the last publish.
// Returns FALSE if the session is not online or the publish fails.
METHOD PublishData : BOOL
VAR_INPUT
	bChangedOnly	: BOOL := FALSE;
END_VAR
IF NOT _ipSession.IsOnline() THEN RETURN; END_IF

_fbDataPayload.Init(ADR(_aDataBuf), SIZEOF(_aDataBuf));
_fbDataPayload.WriteHeader(F_GetUnixTimestampMs(), _ipSession.GetNextSeq());
_writeMetrics(_fbDataPayload, FALSE, bChangedOnly);
PublishData := _ipSession.Publish(_sDataTopic, _fbDataPayload.Buffer, _fbDataPayload.Length, 1, FALSE);

// Sync only the shadows that were written so bChanged stays accurate for any skipped metrics.
IF PublishData THEN
	_syncShadows(bChangedOnly);
END_IF
END_METHOD

// Publishes a DDEATH for this device, signalling the host that it is offline.
// Returns FALSE if the session is not online or the publish fails.
METHOD PublishDeath : BOOL
IF NOT _ipSession.IsOnline() THEN RETURN; END_IF

_fbDeath.Build(F_GetUnixTimestampMs(), _ipSession.GetNextSeq());
PublishDeath := _ipSession.Publish(_sDeathTopic, _fbDeath.Payload.Buffer, _fbDeath.Payload.Length, 1, FALSE);
END_METHOD

// Called by FB_SparkplugSession.AddDevice — stores the device ID and session reference.
// Do not call directly.
METHOD SetSession
VAR_INPUT
	sDeviceId	: STRING(127);
	ipSession	: I_SparkplugSession;
END_VAR
_sDeviceId := sDeviceId;
_ipSession := ipSession;
END_METHOD

// Recomputes bDataPending by comparing each metric's live value against its last-published shadow.
// Floats use deadband comparison; all other types use byte-exact MEMCMP.
// The shadow is NOT updated here — only _syncShadows() writes to it.
METHOD PRIVATE _checkChanges
VAR
	i			: UDINT;
	nSize		: UDINT;
	pStr		: POINTER TO STRING(255);
	pReal		: POINTER TO REAL;
	pLastReal	: POINTER TO REAL;
	pLreal		: POINTER TO LREAL;
	pLastLreal	: POINTER TO LREAL;
END_VAR
bDataPending := FALSE;

FOR i := 0 TO _nMetricCount - 1 DO
	_aMetrics[i].bChanged := FALSE;

	CASE _aMetrics[i].eTypeClass OF
		__SYSTEM.TYPE_CLASS.TYPE_STRING:
			pStr := _aMetrics[i].pValue;
			IF pStr^ <> _aMetrics[i].sLastString THEN
				_aMetrics[i].bChanged := TRUE;
			END_IF

		__SYSTEM.TYPE_CLASS.TYPE_REAL:
			pReal		:= _aMetrics[i].pValue;
			pLastReal	:= ADR(_aMetrics[i].aLastValue);
			IF ABS(pReal^ - pLastReal^) > TO_REAL(_aMetrics[i].fDeadband) THEN
				_aMetrics[i].bChanged := TRUE;
			END_IF

		__SYSTEM.TYPE_CLASS.TYPE_LREAL:
			pLreal		:= _aMetrics[i].pValue;
			pLastLreal	:= ADR(_aMetrics[i].aLastValue);
			IF ABS(pLreal^ - pLastLreal^) > _aMetrics[i].fDeadband THEN
				_aMetrics[i].bChanged := TRUE;
			END_IF
	ELSE
		nSize := _typeSize(_aMetrics[i].eTypeClass);
		IF nSize > 0 AND MEMCMP(_aMetrics[i].pValue, ADR(_aMetrics[i].aLastValue), nSize) <> 0 THEN
			_aMetrics[i].bChanged := TRUE;
		END_IF
	END_CASE

	bDataPending := bDataPending OR _aMetrics[i].bChanged;
END_FOR
END_METHOD

// Returns the byte width of the given IEC type class.
// Returns 0 for STRING (handled separately) and unknown types.
METHOD PRIVATE _typeSize : UDINT
VAR_INPUT
	eTypeClass	: __SYSTEM.TYPE_CLASS;
END_VAR
CASE eTypeClass OF
	__SYSTEM.TYPE_CLASS.TYPE_BOOL,
	__SYSTEM.TYPE_CLASS.TYPE_SINT,
	__SYSTEM.TYPE_CLASS.TYPE_USINT,
	__SYSTEM.TYPE_CLASS.TYPE_BYTE	: _typeSize := 1;
	__SYSTEM.TYPE_CLASS.TYPE_INT,
	__SYSTEM.TYPE_CLASS.TYPE_UINT,
	__SYSTEM.TYPE_CLASS.TYPE_WORD	: _typeSize := 2;
	__SYSTEM.TYPE_CLASS.TYPE_DINT,
	__SYSTEM.TYPE_CLASS.TYPE_UDINT,
	__SYSTEM.TYPE_CLASS.TYPE_DWORD,
	__SYSTEM.TYPE_CLASS.TYPE_REAL	: _typeSize := 4;
	__SYSTEM.TYPE_CLASS.TYPE_LINT,
	__SYSTEM.TYPE_CLASS.TYPE_ULINT,
	__SYSTEM.TYPE_CLASS.TYPE_LWORD,
	__SYSTEM.TYPE_CLASS.TYPE_LREAL	: _typeSize := 8;
ELSE
	_typeSize := 0; // STRING or unknown — handled separately
END_CASE
END_METHOD

// Copies the current live value of every metric into its shadow (last-published record).
// Called after a confirmed DBIRTH or DDATA publish.
METHOD PRIVATE _syncShadows
VAR_INPUT
	bChangedOnly	: BOOL := FALSE;	// when TRUE, only syncs metrics whose bChanged flag is TRUE
END_VAR
VAR
	i		: UDINT;
	nSize	: UDINT;
	pStr	: POINTER TO STRING(255);
END_VAR
FOR i := 0 TO _nMetricCount - 1 DO
	IF bChangedOnly AND NOT _aMetrics[i].bChanged THEN
		;
	ELSIF _aMetrics[i].eTypeClass = __SYSTEM.TYPE_CLASS.TYPE_STRING THEN
		pStr := _aMetrics[i].pValue;
		_aMetrics[i].sLastString := pStr^;
	ELSE
		nSize := _typeSize(_aMetrics[i].eTypeClass);
		IF nSize > 0 THEN
			MEMCPY(ADR(_aMetrics[i].aLastValue), _aMetrics[i].pValue, nSize);
		END_IF
	END_IF
END_FOR
END_METHOD

// Overrides the deadband for a single REAL or LREAL metric identified by its alias.
// Call after AddMetric() and before the first birth cycle.
// Has no effect on non-float metrics (their comparison is always byte-exact).
METHOD SetDeadband
VAR_INPUT
	nAlias		: ULINT;
	fDeadband	: LREAL;
END_VAR
VAR
	i	: UDINT;
END_VAR
FOR i := 0 TO _nMetricCount - 1 DO
	IF _aMetrics[i].nAlias = nAlias THEN
		_aMetrics[i].fDeadband := fDeadband;
		RETURN;
	END_IF
END_FOR
END_METHOD

END_FUNCTION_BLOCK

// ---- Sparkplug/FB_SparkplugSession.TcPOU
// Sparkplug B session manager.
//
// Manages the full Sparkplug lifecycle: MQTT connection, Will registration,
// NBIRTH/NDEATH sequencing, rebirth on command, and reconnection with backoff.
//
// Caller responsibilities:
//   - Declare nBdSeq as RETAIN so it survives power cycles.
//   - Call this FB every PLC cycle regardless of state.
//   - When bBirthRequired rises, publish DBIRTH for every device in the same cycle.
//   - Use GetNextSeq() and Publish() for all outbound data messages.
//
// NOTE: The MQTT client calls (Connect, Subscribe, Publish) target the
// Beckhoff TF6701 Tc3_IotBase FB_IotMqttClient API. Verify method signatures
// against your installed TF6701 version if compile errors occur.

// TODO: support for TLS, certs...
// maybe pass in refrence to MqttClient?
FUNCTION_BLOCK FB_SparkplugSession IMPLEMENTS I_SparkplugSession
VAR_INPUT
	sGroupId		: STRING(127);
	sNodeId			: STRING(127);
	fbMqttClient	: REFERENCE TO FB_IotMqttClient;
	bEnable			: BOOL;
END_VAR
VAR_OUTPUT
	eState			: E_SparkplugState;
	bOnline			: BOOL;
	bBirthRequired	: BOOL;				// TRUE for one cycle — publish DBIRTH on this cycle
	bError			: BOOL;
	sErrorMsg		: STRING(255);
END_VAR
VAR_IN_OUT
	// IMPORTANT: declare this variable as RETAIN in the calling program.
	// It must survive power cycles to satisfy the Sparkplug B specification.
	nBdSeq			: ULINT;
END_VAR
VAR
	_fbNDeath		: FB_NDeathBuilder;
	_fbNBirth		: FB_NBirthBuilder;

	_nSeq			: ULINT;			// 0–255 wrapping; reset to 0 on NBIRTH, 1 after
	_bConnect		: BOOL;

	// Cached topic strings (built once on enable)
	_sNbirthTopic	: STRING(255);
	_sNdeathTopic	: STRING(255);
	_sNcmdTopic		: STRING(255);

	// MQTT Will — must remain stable in memory while the connection is live
	_stWill			: ST_IotMqttWill;

	// Reconnect backoff
	_tReconnect		: TON;

	// One-shot flags
	_bLastEnable		: BOOL;
	_bBirthSignalled	: BOOL;		// TRUE after bBirthRequired was set high this birth cycle
	_bRebirthPending	: BOOL;		// Set by NCMD handler; causes Online→Birthing transition
	_bWasOnline			: BOOL;		// TRUE if connection dropped from Online or Birthing

	// Inbound message processing
	_fbMsg			: FB_IotMqttMessage;
	_fbMsgQueue 	: FB_IotMqttMessageQueue;
	_sMsgTopic		: STRING(255);
	_fbReader		: FB_ProtoReader;
	_fbInnerReader	: FB_ProtoReader;
	_pMetricData	: POINTER TO BYTE;
	_nMetricLen		: UDINT;
	_sMetricName	: STRING(255);
	_bMetricBool	: BOOL;

	// Registered devices — called on each birth cycle
	_aDevices		: ARRAY[0..15] OF I_SparkplugDevice;
	_nDeviceCount	: UDINT;
	_iDev			: UDINT;
END_VAR

fbMqttClient.Execute(_bConnect);

bOnline := (eState = E_SparkplugState.Online);
bError  := fbMqttClient.bError;

// ── State machine ─────────────────────────────────────────────────────────────
CASE eState OF

// ─────────────────────────────────────────────────────────────────────────────
E_SparkplugState.Idle:
	bBirthRequired  := FALSE;
	_bBirthSignalled := FALSE;
	_bWasOnline      := FALSE;

	IF bEnable AND NOT _bLastEnable THEN
		_sNbirthTopic := F_BuildSparkplugTopic(E_SparkplugMessageType.NBIRTH, sGroupId, sNodeId, '');
		_sNdeathTopic := F_BuildSparkplugTopic(E_SparkplugMessageType.NDEATH, sGroupId, sNodeId, '');
		_sNcmdTopic   := F_BuildSparkplugTopic(E_SparkplugMessageType.NCMD,   sGroupId, sNodeId, '');
		sErrorMsg     := '';
		beginConnect();
		eState := E_SparkplugState.Connecting;
	END_IF

// ─────────────────────────────────────────────────────────────────────────────
E_SparkplugState.Connecting:
	IF NOT bEnable THEN
		_bConnect := FALSE;
		eState := E_SparkplugState.Idle;

	ELSIF fbMqttClient.bError THEN
		sErrorMsg := 'Connect failed';
		// bdSeq does NOT increment here — the Will was never registered with a broker
		_tReconnect(IN := FALSE);
		eState := E_SparkplugState.Reconnecting;

	ELSIF fbMqttClient.bConnected THEN
		fbMqttClient.ipMessageQueue := _fbMsgQueue;
		fbMqttClient.Subscribe(_sNcmdTopic, 1);
		eState := E_SparkplugState.Birthing;
	END_IF

// ─────────────────────────────────────────────────────────────────────────────
E_SparkplugState.Birthing:
	IF NOT bEnable OR fbMqttClient.bError OR NOT fbMqttClient.bConnected THEN
		// Connection dropped while birthing — Will has been registered so bdSeq must advance
		nBdSeq := (nBdSeq + 1) MOD 256;
		_bBirthSignalled := FALSE;
		_tReconnect(IN := FALSE);
		IF NOT bEnable THEN
			_bCOnnect := FALSE;
			eState := E_SparkplugState.Idle;
		ELSE
			sErrorMsg := 'Connection lost during birth';
			eState    := E_SparkplugState.Reconnecting;
		END_IF

	ELSIF NOT _bBirthSignalled THEN
		// First half of birth cycle: publish NBIRTH and raise the birth flag
		_nSeq := 0;
		_fbNBirth.Build(F_GetUnixTimestampMs(), nBdSeq);
		fbMqttClient.Publish(
			sTopic       := _sNbirthTopic,
			pPayload     := _fbNBirth.Payload.Buffer,
			nPayloadSize := _fbNBirth.Payload.Length,
			eQos         := TcIotMqttQos.AtLeastOnceDelivery,
			bRetain      := FALSE);
		_nSeq := 1;		// First DBIRTH will use seq=1

		// Publish DBIRTH for every registered device (seq=1, 2, ...)
		IF _nDeviceCount > 0 THEN
			FOR _iDev := 0 TO _nDeviceCount - 1 DO
				IF _aDevices[_iDev] <> 0 THEN
					_aDevices[_iDev].OnBirth();
				END_IF
			END_FOR
		END_IF

		bBirthRequired   := TRUE;	// Signal any external device FBs for one cycle
		_bBirthSignalled := TRUE;

	ELSE
		// Second half: device FBs have had one cycle to see bBirthRequired — go Online
		bBirthRequired   := FALSE;
		_bBirthSignalled := FALSE;
		_bWasOnline      := TRUE;
		eState           := E_SparkplugState.Online;
	END_IF

// ─────────────────────────────────────────────────────────────────────────────
E_SparkplugState.Online:
	IF NOT bEnable THEN
		_bConnect := FALSE;
		nBdSeq := (nBdSeq + 1) MOD 256;
		eState := E_SparkplugState.Idle;

	ELSIF fbMqttClient.bError OR NOT fbMqttClient.bConnected THEN
		sErrorMsg := 'Connection lost';
		nBdSeq    := (nBdSeq + 1) MOD 256;
		_tReconnect(IN := FALSE);
		eState := E_SparkplugState.Reconnecting;

	ELSIF _bRebirthPending THEN
		// Soft rebirth (triggered by NCMD or STATE recovery) — bdSeq does NOT change
		_bRebirthPending := FALSE;
		_bBirthSignalled := FALSE;
		eState           := E_SparkplugState.Birthing;

	ELSE
		pollMessages();
	END_IF

// ─────────────────────────────────────────────────────────────────────────────
E_SparkplugState.Reconnecting:
	_tReconnect(IN := TRUE, PT := T#5S);

	IF NOT bEnable THEN
		_tReconnect(IN := FALSE);
		eState := E_SparkplugState.Idle;

	ELSIF _tReconnect.Q THEN
		_tReconnect(IN := FALSE);
		beginConnect();
		eState := E_SparkplugState.Connecting;
	END_IF

END_CASE

_bLastEnable := bEnable;

// Registers a device FB with the session.
// The session will call ipDevice.OnBirth() automatically on every birth cycle.
// Call once during startup after AddMetric(), before the first birth cycle.
METHOD AddDevice
VAR_INPUT
	sDeviceId	: STRING(127);
	ipDevice	: I_SparkplugDevice;
END_VAR
VAR
	ipMe	: I_SparkplugSession;
END_VAR
IF _nDeviceCount >= 16 THEN RETURN; END_IF

ipMe := THIS^;
ipDevice.SetSession(sDeviceId, ipMe);
_aDevices[_nDeviceCount] := ipDevice;
_nDeviceCount := _nDeviceCount + 1;
END_METHOD

// Builds the NDEATH Will payload from the current nBdSeq, then initiates
// the MQTT connection. nBdSeq must already be at the correct value for this
// connection before this method is called.
METHOD PRIVATE beginConnect
// Build NDEATH — this becomes the MQTT Will payload.
// The broker will publish it automatically on ungraceful disconnect.
_fbNDeath.Build(nBdSeq);

_stWill.sTopic			:= _sNdeathTopic;
_stWill.pPayload     	:= _fbNDeath.PayloadBuffer;
_stWill.nPayloadSize 	:= _fbNDeath.PayloadLength;
_stWill.eQos         	:= TcIotMqttQos.AtLeastOnceDelivery;
_stWill.bRetain      	:= FALSE;

fbMqttClient.stWill 		:= _stWill;

_bConnect := TRUE;
END_METHOD

// Returns the current seq value and advances the counter (0–255 wrapping).
// Device FBs must call this once per published message to stamp the payload header.
METHOD GetNextSeq : ULINT
GetNextSeq := _nSeq;
_nSeq      := (_nSeq + 1) MOD 256;
END_METHOD

// Returns the Sparkplug group ID configured on this session.
// Device FBs use this to build their own topics without duplicating the group/node at the call site.
PROPERTY GroupId : STRING(127)
GET
GroupId := sGroupId;
END_GET
END_PROPERTY

// Parses an NCMD payload. Sets _bRebirthPending if Node Control/Rebirth = TRUE.
// All other node commands are ignored here; device DCMDs are handled by device FBs.
METHOD PRIVATE handleNcmd
VAR_INPUT
	pPayload	: PVOID;
	nLen		: UDINT;
END_VAR
VAR
	pMetric		: POINTER TO BYTE;
	nMetricLen	: UDINT;
	sName		: STRING(255);
	bBoolVal	: BOOL;
	bGotName	: BOOL;
	bGotBool	: BOOL;
END_VAR
// Decode the outer Payload message — we only care about Metric entries (field 2)
_fbReader.Init(pPayload, nLen);
WHILE _fbReader.Next() DO
	IF _fbReader.FieldNumber = 2 THEN
		_fbReader.ReadBytes(pData => pMetric, nLen => nMetricLen);

		// Decode the inner Metric message
		sName    := '';
		bBoolVal := FALSE;
		bGotName := FALSE;
		bGotBool := FALSE;

		_fbInnerReader.Init(pMetric, nMetricLen);
		WHILE _fbInnerReader.Next() DO
			CASE _fbInnerReader.FieldNumber OF
				1:	// name
					_fbInnerReader.ReadString(sValue => sName);
					bGotName := TRUE;
				14:	// boolean_value
					_fbInnerReader.ReadBool(bValue => bBoolVal);
					bGotBool := TRUE;
			ELSE
				_fbInnerReader.Skip();
			END_CASE
		END_WHILE

		IF bGotName AND bGotBool
			AND sName = 'Node Control/Rebirth'
			AND bBoolVal
		THEN
			_bRebirthPending := TRUE;
		END_IF
	ELSE
		_fbReader.Skip();
	END_IF
END_WHILE
END_METHOD

// Returns TRUE when the session is in the Online state.
// Implements I_SparkplugSession — avoids naming conflict with the bOnline VAR_OUTPUT.
METHOD IsOnline : BOOL
IsOnline := bOnline;
END_METHOD

// Returns the Sparkplug node ID configured on this session.
// Device FBs use this to build their own topics without duplicating the group/node at the call site.
PROPERTY NodeId : STRING(127)
GET
NodeId := sNodeId;
END_GET
END_PROPERTY

// Drains the inbound message queue for this cycle.
// Dispatches NCMD messages to handleNcmd; all other topics are silently discarded.
METHOD PRIVATE pollMessages
// Drain one message per cycle.
// The Sparkplug B spec requires the primary application to send NCMD/rebirth
// to edge nodes after it reconnects, so rebirth is driven by NCMD only.
IF _fbMsgQueue.nQueuedMessages > 0 AND _fbMsgQueue.Dequeue(_fbMsg) THEN
	_fbMsg.GetTopic(ADR(_sMsgTopic), 255);
	IF _sMsgTopic = _sNcmdTopic THEN
		handleNcmd(_fbMsg.pPayload, _fbMsg.nPayloadSize);
	END_IF
END_IF
END_METHOD

// Publishes a pre-encoded payload. Device FBs use this to send DBIRTH and DDATA.
// Only call when bOnline is TRUE or bBirthRequired is TRUE.
METHOD Publish : BOOL
VAR_INPUT
	sTopic		: STRING(255);
	pPayload	: POINTER TO BYTE;
	nLen		: UDINT;
	nQos		: UDINT := 1;
	bRetain		: BOOL  := FALSE;
END_VAR
IF eState = E_SparkplugState.Online OR eState = E_SparkplugState.Birthing THEN
	Publish := fbMqttClient.Publish(
		sTopic       := sTopic,
		pPayload     := pPayload,
		nPayloadSize := nLen,
		eQos         := UDINT_TO_SINT(nQos),
		bRetain      := bRetain);
END_IF
END_METHOD

END_FUNCTION_BLOCK

// ---- Tests/F_Assert.TcPOU
// Increments nPass if bCondition is TRUE, otherwise increments nFail and records
// the name of the first failure in sFirstFail.
FUNCTION F_Assert : BOOL
VAR_INPUT
	bCondition	: BOOL;
	sTestName	: STRING(255);
END_VAR
VAR_IN_OUT
	nPass		: UDINT;
	nFail		: UDINT;
	sFirstFail	: STRING(255);
END_VAR

IF bCondition THEN
	nPass    := nPass + 1;
	F_Assert := TRUE;
ELSE
	nFail := nFail + 1;
	IF nFail = 1 THEN
		sFirstFail := sTestName;
	END_IF
	F_Assert := FALSE;
END_IF

END_FUNCTION

// ---- Tests/PRG_ProtoTests.TcPOU
// Proto round-trip test suite.
// Set bRun := TRUE to execute. Results appear in nPass, nFail, bAllPassed, sFirstFail.
PROGRAM PRG_ProtoTests
VAR
	// Trigger
	bRun		: BOOL;
	_bLastRun	: BOOL;

	// Results
	nPass		: UDINT;
	nFail		: UDINT;
	bAllPassed	: BOOL;
	sFirstFail	: STRING(255);
	bRan		: BOOL;

	// Shared writer / reader
	fbW			: FB_ProtoWriter;
	fbR			: FB_ProtoReader;

	// Second writer for nested-message test
	fbWInner	: FB_ProtoWriter;

	// Buffers
	aBuf		: ARRAY[0..511] OF BYTE;
	aBufInner	: ARRAY[0..63]  OF BYTE;
	aSmallBuf	: ARRAY[0..3]   OF BYTE;   // intentionally tiny for overflow test

	// Known byte sequence used in the Bytes test
	aTestBytes	: ARRAY[0..3] OF BYTE := [16#DE, 16#AD, 16#BE, 16#EF];

	// Readback variables
	nU32		: UDINT;
	nU64		: ULINT;
	bVal		: BOOL;
	fVal		: REAL;
	dVal		: LREAL;
	sVal		: STRING(255);
	pBytes		: POINTER TO BYTE;
	nBytesLen	: UDINT;
END_VAR

// Run once per rising edge of bRun
IF NOT (bRun AND NOT _bLastRun) THEN
	_bLastRun := bRun;
	RETURN;
END_IF
_bLastRun := bRun;

nPass      := 0;
nFail      := 0;
sFirstFail := '';
bRan       := FALSE;

// ── T01: UInt32 — single-byte varint (value fits in 7 bits) ──────────────────
fbW.Init(ADR(aBuf), SIZEOF(aBuf));
fbW.WriteUInt32(1, 5);
fbR.Init(ADR(aBuf), fbW.Length);
fbR.Next();
fbR.ReadUInt32(nValue => nU32);
F_Assert(
	bCondition := fbR.FieldNumber = 1 AND nU32 = 5 AND NOT fbR.HasError,
	sTestName  := 'T01 UInt32 single-byte varint',
	nPass := nPass, nFail := nFail, sFirstFail := sFirstFail);

// ── T02: UInt32 — multi-byte varint (value > 127, needs 2 bytes) ─────────────
fbW.Init(ADR(aBuf), SIZEOF(aBuf));
fbW.WriteUInt32(2, 300);
fbR.Init(ADR(aBuf), fbW.Length);
fbR.Next();
fbR.ReadUInt32(nValue => nU32);
F_Assert(
	bCondition := fbR.FieldNumber = 2 AND nU32 = 300 AND NOT fbR.HasError,
	sTestName  := 'T02 UInt32 multi-byte varint',
	nPass := nPass, nFail := nFail, sFirstFail := sFirstFail);

// ── T03: UInt64 — Sparkplug-realistic timestamp (10-byte varint) ─────────────
fbW.Init(ADR(aBuf), SIZEOF(aBuf));
fbW.WriteUInt64(3, 1700000000000);
fbR.Init(ADR(aBuf), fbW.Length);
fbR.Next();
fbR.ReadUInt64(nValue => nU64);
F_Assert(
	bCondition := fbR.FieldNumber = 3 AND nU64 = 1700000000000 AND NOT fbR.HasError,
	sTestName  := 'T03 UInt64 large value',
	nPass := nPass, nFail := nFail, sFirstFail := sFirstFail);

// ── T04: Bool TRUE ────────────────────────────────────────────────────────────
fbW.Init(ADR(aBuf), SIZEOF(aBuf));
fbW.WriteBool(4, TRUE);
fbR.Init(ADR(aBuf), fbW.Length);
fbR.Next();
fbR.ReadBool(bValue => bVal);
F_Assert(
	bCondition := fbR.FieldNumber = 4 AND bVal = TRUE AND NOT fbR.HasError,
	sTestName  := 'T04 Bool TRUE',
	nPass := nPass, nFail := nFail, sFirstFail := sFirstFail);

// ── T05: Bool FALSE ───────────────────────────────────────────────────────────
fbW.Init(ADR(aBuf), SIZEOF(aBuf));
fbW.WriteBool(5, FALSE);
fbR.Init(ADR(aBuf), fbW.Length);
fbR.Next();
fbR.ReadBool(bValue => bVal);
F_Assert(
	bCondition := fbR.FieldNumber = 5 AND bVal = FALSE AND NOT fbR.HasError,
	sTestName  := 'T05 Bool FALSE',
	nPass := nPass, nFail := nFail, sFirstFail := sFirstFail);

// ── T06: Float (Fixed32 wire type) ───────────────────────────────────────────
// 1.5 is exactly representable in IEEE 754 — safe for exact equality check.
fbW.Init(ADR(aBuf), SIZEOF(aBuf));
fbW.WriteFloat(6, 1.5);
fbR.Init(ADR(aBuf), fbW.Length);
fbR.Next();
fbR.ReadFloat(fValue => fVal);
F_Assert(
	bCondition := fbR.FieldNumber = 6 AND fVal = 1.5 AND NOT fbR.HasError,
	sTestName  := 'T06 Float round-trip',
	nPass := nPass, nFail := nFail, sFirstFail := sFirstFail);

// ── T07: Double (Fixed64 wire type) ──────────────────────────────────────────
// 0.125 = 2^-3, exactly representable.
fbW.Init(ADR(aBuf), SIZEOF(aBuf));
fbW.WriteDouble(7, 0.125);
fbR.Init(ADR(aBuf), fbW.Length);
fbR.Next();
fbR.ReadDouble(fValue => dVal);
F_Assert(
	bCondition := fbR.FieldNumber = 7 AND dVal = 0.125 AND NOT fbR.HasError,
	sTestName  := 'T07 Double round-trip',
	nPass := nPass, nFail := nFail, sFirstFail := sFirstFail);

// ── T08: String ───────────────────────────────────────────────────────────────
fbW.Init(ADR(aBuf), SIZEOF(aBuf));
fbW.WriteString(8, 'hello');
fbR.Init(ADR(aBuf), fbW.Length);
fbR.Next();
fbR.ReadString(sValue => sVal);
F_Assert(
	bCondition := fbR.FieldNumber = 8 AND sVal = 'hello' AND NOT fbR.HasError,
	sTestName  := 'T08 String round-trip',
	nPass := nPass, nFail := nFail, sFirstFail := sFirstFail);

// ── T09: Bytes ────────────────────────────────────────────────────────────────
fbW.Init(ADR(aBuf), SIZEOF(aBuf));
fbW.WriteBytes(9, ADR(aTestBytes), SIZEOF(aTestBytes));
fbR.Init(ADR(aBuf), fbW.Length);
fbR.Next();
fbR.ReadBytes(pData => pBytes, nLen => nBytesLen);
F_Assert(
	bCondition := fbR.FieldNumber = 9
		AND nBytesLen = 4
		AND pBytes[0] = 16#DE AND pBytes[1] = 16#AD
		AND pBytes[2] = 16#BE AND pBytes[3] = 16#EF
		AND NOT fbR.HasError,
	sTestName  := 'T09 Bytes round-trip',
	nPass := nPass, nFail := nFail, sFirstFail := sFirstFail);

// ── T10: Multiple fields written and read in sequence ─────────────────────────
fbW.Init(ADR(aBuf), SIZEOF(aBuf));
fbW.WriteUInt32(1, 42);
fbW.WriteBool(2, TRUE);
fbW.WriteFloat(3, 1.5);
fbR.Init(ADR(aBuf), fbW.Length);

fbR.Next(); fbR.ReadUInt32(nValue => nU32);
F_Assert(
	bCondition := fbR.FieldNumber = 1 AND nU32 = 42,
	sTestName  := 'T10a Multi-field field 1',
	nPass := nPass, nFail := nFail, sFirstFail := sFirstFail);

fbR.Next(); fbR.ReadBool(bValue => bVal);
F_Assert(
	bCondition := fbR.FieldNumber = 2 AND bVal = TRUE,
	sTestName  := 'T10b Multi-field field 2',
	nPass := nPass, nFail := nFail, sFirstFail := sFirstFail);

fbR.Next(); fbR.ReadFloat(fValue => fVal);
F_Assert(
	bCondition := fbR.FieldNumber = 3 AND fVal = 1.5,
	sTestName  := 'T10c Multi-field field 3',
	nPass := nPass, nFail := nFail, sFirstFail := sFirstFail);

F_Assert(
	bCondition := NOT fbR.Next(),
	sTestName  := 'T10d Multi-field end of buffer',
	nPass := nPass, nFail := nFail, sFirstFail := sFirstFail);

// ── T11: Skip ────────────────────────────────────────────────────────────────
// Write fields 1 and 3; skip field 1 and verify field 3 is read correctly.
fbW.Init(ADR(aBuf), SIZEOF(aBuf));
fbW.WriteUInt32(1, 99);
fbW.WriteFloat(2, 2.5);    // Fixed32 — exercises Skip for that wire type too
fbW.WriteUInt32(3, 77);
fbR.Init(ADR(aBuf), fbW.Length);

fbR.Next(); fbR.Skip();   // skip UInt32
fbR.Next(); fbR.Skip();   // skip Float
fbR.Next(); fbR.ReadUInt32(nValue => nU32);
F_Assert(
	bCondition := fbR.FieldNumber = 3 AND nU32 = 77 AND NOT fbR.HasError,
	sTestName  := 'T11 Skip fields',
	nPass := nPass, nFail := nFail, sFirstFail := sFirstFail);

// ── T12: Nested message — minimal Sparkplug Metric inside a Payload ───────────
// Inner: Metric { alias=1 (f2), datatype=11/Boolean (f4), boolean_value=true (f14) }
fbWInner.Init(ADR(aBufInner), SIZEOF(aBufInner));
fbWInner.WriteUInt64(2,  1);    // alias
fbWInner.WriteUInt32(4, 11);    // datatype = Boolean
fbWInner.WriteBool(14, TRUE);   // boolean_value

// Outer: Payload { timestamp (f1), metrics (f2) }
fbW.Init(ADR(aBuf), SIZEOF(aBuf));
fbW.WriteUInt64(1, 1700000000000);
fbW.WriteBytes(2, ADR(aBufInner), fbWInner.Length);

// Decode outer payload
fbR.Init(ADR(aBuf), fbW.Length);
fbR.Next(); fbR.ReadUInt64(nValue => nU64);
F_Assert(
	bCondition := fbR.FieldNumber = 1 AND nU64 = 1700000000000,
	sTestName  := 'T12a Nested outer timestamp',
	nPass := nPass, nFail := nFail, sFirstFail := sFirstFail);

fbR.Next(); fbR.ReadBytes(pData => pBytes, nLen => nBytesLen);
F_Assert(
	bCondition := fbR.FieldNumber = 2 AND nBytesLen = fbWInner.Length AND NOT fbR.HasError,
	sTestName  := 'T12b Nested metrics field',
	nPass := nPass, nFail := nFail, sFirstFail := sFirstFail);

// Re-use fbR to decode the inner metric bytes (zero-copy — pBytes points into aBuf)
fbR.Init(pBytes, nBytesLen);

fbR.Next(); fbR.ReadUInt64(nValue => nU64);
F_Assert(
	bCondition := fbR.FieldNumber = 2 AND nU64 = 1,
	sTestName  := 'T12c Nested metric alias',
	nPass := nPass, nFail := nFail, sFirstFail := sFirstFail);

fbR.Next(); fbR.ReadUInt32(nValue => nU32);
F_Assert(
	bCondition := fbR.FieldNumber = 4 AND nU32 = 11,
	sTestName  := 'T12d Nested metric datatype',
	nPass := nPass, nFail := nFail, sFirstFail := sFirstFail);

fbR.Next(); fbR.ReadBool(bValue => bVal);
F_Assert(
	bCondition := fbR.FieldNumber = 14 AND bVal = TRUE AND NOT fbR.HasError,
	sTestName  := 'T12e Nested metric boolean_value',
	nPass := nPass, nFail := nFail, sFirstFail := sFirstFail);

// ── T13: Writer overflow ──────────────────────────────────────────────────────
// aSmallBuf is 4 bytes; a UInt64 field for 1700000000000 encodes to 11 bytes.
fbW.Init(ADR(aSmallBuf), SIZEOF(aSmallBuf));
fbW.WriteUInt64(1, 1700000000000);
F_Assert(
	bCondition := fbW.HasError,
	sTestName  := 'T13 Writer overflow sets HasError',
	nPass := nPass, nFail := nFail, sFirstFail := sFirstFail);

// ── T14: Reader wire type mismatch ───────────────────────────────────────────
// Field is encoded as Fixed32 (Float); reading it as Varint (UInt32) must error.
fbW.Init(ADR(aBuf), SIZEOF(aBuf));
fbW.WriteFloat(1, 1.5);
fbR.Init(ADR(aBuf), fbW.Length);
fbR.Next();
fbR.ReadUInt32(nValue => nU32);   // wrong read type
F_Assert(
	bCondition := fbR.HasError,
	sTestName  := 'T14 Reader wire type mismatch sets HasError',
	nPass := nPass, nFail := nFail, sFirstFail := sFirstFail);

// ── Done ─────────────────────────────────────────────────────────────────────
bAllPassed := (nFail = 0);
bRan       := TRUE;

END_PROGRAM

// ---- Tests/PRG_SparkplugPayloadTests.TcPOU
// Sparkplug payload builder test suite.
// Set bRun := TRUE to execute. Results in nPass, nFail, bAllPassed, sFirstFail.
PROGRAM PRG_SparkplugPayloadTests
VAR
	bRun		: BOOL;
	_bLastRun	: BOOL;

	nPass		: UDINT;
	nFail		: UDINT;
	bAllPassed	: BOOL;
	sFirstFail	: STRING(255);
	bRan		: BOOL;

	// Builders under test
	fbNDeath	: FB_NDeathBuilder;
	fbNBirth	: FB_NBirthBuilder;
	fbDDeath	: FB_DDeathBuilder;

	// Generic payload builder for metric writer tests
	aBuf		: ARRAY[0..511] OF BYTE;
	fbPayload	: FB_SparkplugPayload;

	// Readers
	fbR			: FB_ProtoReader;
	fbRInner	: FB_ProtoReader;

	// Readback vars
	nU32		: UDINT;
	nU64		: ULINT;
	bVal		: BOOL;
	fVal		: REAL;
	dVal		: LREAL;
	sVal		: STRING(255);
	pMetric		: POINTER TO BYTE;
	nMetricLen	: UDINT;

	// Fixed test values
	nTestTs		: ULINT := 1700000000000;	// ms — a Sparkplug-realistic timestamp
	nTestBdSeq	: ULINT := 42;
	nTestSeq	: ULINT := 7;
END_VAR

IF NOT (bRun AND NOT _bLastRun) THEN
	_bLastRun := bRun;
	RETURN;
END_IF
_bLastRun := bRun;

nPass      := 0;
nFail      := 0;
sFirstFail := '';
bRan       := FALSE;

// ════════════════════════════════════════════════════════════════════════════
// GROUP 1 — F_BuildSparkplugTopic
// ════════════════════════════════════════════════════════════════════════════

// T01: Node-level topic — no device ID
F_Assert(
	bCondition := F_BuildSparkplugTopic(E_SparkplugMessageType.NBIRTH, 'Grp', 'Node', '') = 'spBv1.0/Grp/NBIRTH/Node',
	sTestName  := 'T01 Topic node-level NBIRTH',
	nPass := nPass, nFail := nFail, sFirstFail := sFirstFail);

// T02: Device-level topic — device ID appended
F_Assert(
	bCondition := F_BuildSparkplugTopic(E_SparkplugMessageType.DDATA, 'G', 'N', 'D') = 'spBv1.0/G/DDATA/N/D',
	sTestName  := 'T02 Topic device-level DDATA',
	nPass := nPass, nFail := nFail, sFirstFail := sFirstFail);

// T03: NCMD node-level
F_Assert(
	bCondition := F_BuildSparkplugTopic(E_SparkplugMessageType.NCMD, 'Plant1', 'PLC1', '') = 'spBv1.0/Plant1/NCMD/PLC1',
	sTestName  := 'T03 Topic NCMD',
	nPass := nPass, nFail := nFail, sFirstFail := sFirstFail);

// T04: NDEATH
F_Assert(
	bCondition := F_BuildSparkplugTopic(E_SparkplugMessageType.NDEATH, 'Grp', 'Node', '') = 'spBv1.0/Grp/NDEATH/Node',
	sTestName  := 'T04 Topic NDEATH',
	nPass := nPass, nFail := nFail, sFirstFail := sFirstFail);


// ════════════════════════════════════════════════════════════════════════════
// GROUP 2 — FB_NDeathBuilder
// Expected outer payload: f2 (metric) only — no timestamp, no seq.
// Expected inner metric:  f1=name, f4=datatype, f11=long_value
// ════════════════════════════════════════════════════════════════════════════

fbNDeath.Build(nTestBdSeq);
fbR.Init(fbNDeath.PayloadBuffer, fbNDeath.PayloadLength);

// T05: builder reports no error
F_Assert(
	bCondition := fbNDeath.IsValid,
	sTestName  := 'T05 NDeathBuilder IsValid',
	nPass := nPass, nFail := nFail, sFirstFail := sFirstFail);

// T06: first (and only) outer field is the metrics field (f2) — no timestamp or seq
fbR.Next();
F_Assert(
	bCondition := fbR.FieldNumber = 2,
	sTestName  := 'T06 NDEATH outer field is metrics (f2), no header fields',
	nPass := nPass, nFail := nFail, sFirstFail := sFirstFail);

// T07–T10: decode the inner bdSeq metric
fbR.ReadBytes(pData => pMetric, nLen => nMetricLen);
fbRInner.Init(pMetric, nMetricLen);

fbRInner.Next(); fbRInner.ReadString(sValue => sVal);
F_Assert(
	bCondition := fbRInner.FieldNumber = 1 AND sVal = 'bdSeq',
	sTestName  := 'T07 NDEATH metric name = bdSeq',
	nPass := nPass, nFail := nFail, sFirstFail := sFirstFail);

fbRInner.Next(); fbRInner.ReadUInt32(nValue => nU32);
F_Assert(
	bCondition := fbRInner.FieldNumber = 4 AND nU32 = TO_UDINT(E_SparkplugDataType.UInt64),
	sTestName  := 'T08 NDEATH metric datatype = UInt64',
	nPass := nPass, nFail := nFail, sFirstFail := sFirstFail);

fbRInner.Next(); fbRInner.ReadUInt64(nValue => nU64);
F_Assert(
	bCondition := fbRInner.FieldNumber = 11 AND nU64 = nTestBdSeq,
	sTestName  := 'T09 NDEATH metric long_value = bdSeq',
	nPass := nPass, nFail := nFail, sFirstFail := sFirstFail);

F_Assert(
	bCondition := NOT fbRInner.Next() AND NOT fbR.Next(),
	sTestName  := 'T10 NDEATH no extra fields in metric or payload',
	nPass := nPass, nFail := nFail, sFirstFail := sFirstFail);


// ════════════════════════════════════════════════════════════════════════════
// GROUP 3 — FB_NBirthBuilder
// Expected outer payload: f1=timestamp, f3=seq(0), f2=bdSeq metric, f2=Rebirth metric
// bdSeq metric inner:    f1=name, f4=datatype, f11=long_value  (no alias: alias=0)
// Rebirth metric inner:  f1=name, f4=datatype, f14=boolean_value
// ════════════════════════════════════════════════════════════════════════════

fbNBirth.Build(nTestTs, nTestBdSeq);
fbR.Init(fbNBirth.Payload.Buffer, fbNBirth.Payload.Length);

// T11: builder reports no error
F_Assert(
	bCondition := NOT fbNBirth.Payload.HasError,
	sTestName  := 'T11 NBirthBuilder no error',
	nPass := nPass, nFail := nFail, sFirstFail := sFirstFail);

// T12–T13: outer header
fbR.Next(); fbR.ReadUInt64(nValue => nU64);
F_Assert(
	bCondition := fbR.FieldNumber = 1 AND nU64 = nTestTs,
	sTestName  := 'T12 NBIRTH timestamp correct',
	nPass := nPass, nFail := nFail, sFirstFail := sFirstFail);

fbR.Next(); fbR.ReadUInt64(nValue => nU64);
F_Assert(
	bCondition := fbR.FieldNumber = 3 AND nU64 = 0,
	sTestName  := 'T13 NBIRTH seq = 0',
	nPass := nPass, nFail := nFail, sFirstFail := sFirstFail);

// T14–T16: first metric — bdSeq
fbR.Next(); fbR.ReadBytes(pData => pMetric, nLen => nMetricLen);
F_Assert(
	bCondition := fbR.FieldNumber = 2,
	sTestName  := 'T14 NBIRTH first metric field present',
	nPass := nPass, nFail := nFail, sFirstFail := sFirstFail);

fbRInner.Init(pMetric, nMetricLen);
fbRInner.Next(); fbRInner.ReadString(sValue => sVal);
F_Assert(
	bCondition := fbRInner.FieldNumber = 1 AND sVal = 'bdSeq',
	sTestName  := 'T15 NBIRTH bdSeq metric name',
	nPass := nPass, nFail := nFail, sFirstFail := sFirstFail);

fbRInner.Next(); fbRInner.ReadUInt32(nValue => nU32);
fbRInner.Next(); fbRInner.ReadUInt64(nValue => nU64);
F_Assert(
	bCondition := nU32 = TO_UDINT(E_SparkplugDataType.UInt64) AND nU64 = nTestBdSeq,
	sTestName  := 'T16 NBIRTH bdSeq metric datatype and value',
	nPass := nPass, nFail := nFail, sFirstFail := sFirstFail);

// T17–T19: second metric — Node Control/Rebirth
fbR.Next(); fbR.ReadBytes(pData => pMetric, nLen => nMetricLen);
F_Assert(
	bCondition := fbR.FieldNumber = 2,
	sTestName  := 'T17 NBIRTH second metric field present',
	nPass := nPass, nFail := nFail, sFirstFail := sFirstFail);

fbRInner.Init(pMetric, nMetricLen);
fbRInner.Next(); fbRInner.ReadString(sValue => sVal);
F_Assert(
	bCondition := fbRInner.FieldNumber = 1 AND sVal = 'Node Control/Rebirth',
	sTestName  := 'T18 NBIRTH Rebirth metric name',
	nPass := nPass, nFail := nFail, sFirstFail := sFirstFail);

fbRInner.Next(); fbRInner.ReadUInt32(nValue => nU32);
fbRInner.Next(); fbRInner.ReadBool(bValue => bVal);
F_Assert(
	bCondition := nU32 = TO_UDINT(E_SparkplugDataType.Boolean) AND bVal = FALSE,
	sTestName  := 'T19 NBIRTH Rebirth metric datatype and value=FALSE',
	nPass := nPass, nFail := nFail, sFirstFail := sFirstFail);

F_Assert(
	bCondition := NOT fbR.Next(),
	sTestName  := 'T20 NBIRTH no extra outer fields',
	nPass := nPass, nFail := nFail, sFirstFail := sFirstFail);


// ════════════════════════════════════════════════════════════════════════════
// GROUP 4 — FB_DDeathBuilder
// Expected outer payload: f1=timestamp, f3=seq — no metrics follow.
// ════════════════════════════════════════════════════════════════════════════

fbDDeath.Build(nTestTs, nTestSeq);
fbR.Init(fbDDeath.Payload.Buffer, fbDDeath.Payload.Length);

fbR.Next(); fbR.ReadUInt64(nValue => nU64);
F_Assert(
	bCondition := fbR.FieldNumber = 1 AND nU64 = nTestTs,
	sTestName  := 'T21 DDEATH timestamp correct',
	nPass := nPass, nFail := nFail, sFirstFail := sFirstFail);

fbR.Next(); fbR.ReadUInt64(nValue => nU64);
F_Assert(
	bCondition := fbR.FieldNumber = 3 AND nU64 = nTestSeq,
	sTestName  := 'T22 DDEATH seq correct',
	nPass := nPass, nFail := nFail, sFirstFail := sFirstFail);

F_Assert(
	bCondition := NOT fbR.Next(),
	sTestName  := 'T23 DDEATH no metrics',
	nPass := nPass, nFail := nFail, sFirstFail := sFirstFail);


// ════════════════════════════════════════════════════════════════════════════
// GROUP 5 — FB_SparkplugPayload metric writers
// Helper pattern for each test:
//   Init → WriteHeader → WriteXxxMetric → decode outer (skip f1+f4) → decode inner
// ════════════════════════════════════════════════════════════════════════════

// ── T24–T27: WriteBoolMetric — birth mode (name + alias + datatype + value) ─
fbPayload.Init(ADR(aBuf), SIZEOF(aBuf));
fbPayload.WriteHeader(nTestTs, 0);
fbPayload.WriteBoolMetric('Running', 1, E_SparkplugDataType.Boolean, TRUE);

fbR.Init(fbPayload.Buffer, fbPayload.Length);
fbR.Next(); fbR.Skip();		// f1: timestamp
fbR.Next(); fbR.Skip();		// f3: seq
fbR.Next(); fbR.ReadBytes(pData => pMetric, nLen => nMetricLen);

fbRInner.Init(pMetric, nMetricLen);
fbRInner.Next(); fbRInner.ReadString(sValue => sVal);
F_Assert(
	bCondition := fbRInner.FieldNumber = 1 AND sVal = 'Running',
	sTestName  := 'T24 WriteBoolMetric name',
	nPass := nPass, nFail := nFail, sFirstFail := sFirstFail);

fbRInner.Next(); fbRInner.ReadUInt64(nValue => nU64);
F_Assert(
	bCondition := fbRInner.FieldNumber = 2 AND nU64 = 1,
	sTestName  := 'T25 WriteBoolMetric alias',
	nPass := nPass, nFail := nFail, sFirstFail := sFirstFail);

fbRInner.Next(); fbRInner.ReadUInt32(nValue => nU32);
F_Assert(
	bCondition := fbRInner.FieldNumber = 4 AND nU32 = TO_UDINT(E_SparkplugDataType.Boolean),
	sTestName  := 'T26 WriteBoolMetric datatype',
	nPass := nPass, nFail := nFail, sFirstFail := sFirstFail);

fbRInner.Next(); fbRInner.ReadBool(bValue => bVal);
F_Assert(
	bCondition := fbRInner.FieldNumber = 14 AND bVal = TRUE,
	sTestName  := 'T27 WriteBoolMetric value',
	nPass := nPass, nFail := nFail, sFirstFail := sFirstFail);

// ── T28–T29: WriteBoolMetric — data mode (no name; first field must be alias) ─
fbPayload.Init(ADR(aBuf), SIZEOF(aBuf));
fbPayload.WriteHeader(nTestTs, 5);
fbPayload.WriteBoolMetric('', 3, E_SparkplugDataType.Boolean, FALSE);

fbR.Init(fbPayload.Buffer, fbPayload.Length);
fbR.Next(); fbR.Skip();
fbR.Next(); fbR.Skip();
fbR.Next(); fbR.ReadBytes(pData => pMetric, nLen => nMetricLen);

fbRInner.Init(pMetric, nMetricLen);
fbRInner.Next();
F_Assert(
	bCondition := fbRInner.FieldNumber = 2,
	sTestName  := 'T28 WriteBoolMetric data mode: first field is alias (no name)',
	nPass := nPass, nFail := nFail, sFirstFail := sFirstFail);
fbRInner.ReadUInt64(nValue => nU64);
F_Assert(
	bCondition := nU64 = 3,
	sTestName  := 'T29 WriteBoolMetric data mode: alias value correct',
	nPass := nPass, nFail := nFail, sFirstFail := sFirstFail);

// ── T30–T31: WriteUInt32Metric (int_value → proto field 10) ─────────────────
fbPayload.Init(ADR(aBuf), SIZEOF(aBuf));
fbPayload.WriteHeader(nTestTs, 0);
fbPayload.WriteUInt32Metric('Speed', 2, E_SparkplugDataType.UInt32, 1500);

fbR.Init(fbPayload.Buffer, fbPayload.Length);
fbR.Next(); fbR.Skip(); fbR.Next(); fbR.Skip();
fbR.Next(); fbR.ReadBytes(pData => pMetric, nLen => nMetricLen);

fbRInner.Init(pMetric, nMetricLen);
fbRInner.Next(); fbRInner.Skip();		// f1: name
fbRInner.Next(); fbRInner.Skip();		// f2: alias
fbRInner.Next(); fbRInner.ReadUInt32(nValue => nU32);
F_Assert(
	bCondition := fbRInner.FieldNumber = 4 AND nU32 = TO_UDINT(E_SparkplugDataType.UInt32),
	sTestName  := 'T30 WriteUInt32Metric datatype',
	nPass := nPass, nFail := nFail, sFirstFail := sFirstFail);

fbRInner.Next(); fbRInner.ReadUInt32(nValue => nU32);
F_Assert(
	bCondition := fbRInner.FieldNumber = 10 AND nU32 = 1500,
	sTestName  := 'T31 WriteUInt32Metric int_value (f10)',
	nPass := nPass, nFail := nFail, sFirstFail := sFirstFail);

// ── T32–T33: WriteFloatMetric (float_value → proto field 12) ────────────────
fbPayload.Init(ADR(aBuf), SIZEOF(aBuf));
fbPayload.WriteHeader(nTestTs, 0);
fbPayload.WriteFloatMetric('Temp', 3, E_SparkplugDataType.Float, 2.5);

fbR.Init(fbPayload.Buffer, fbPayload.Length);
fbR.Next(); fbR.Skip(); fbR.Next(); fbR.Skip();
fbR.Next(); fbR.ReadBytes(pData => pMetric, nLen => nMetricLen);

fbRInner.Init(pMetric, nMetricLen);
fbRInner.Next(); fbRInner.Skip();		// f1: name
fbRInner.Next(); fbRInner.Skip();		// f2: alias
fbRInner.Next(); fbRInner.ReadUInt32(nValue => nU32);
F_Assert(
	bCondition := fbRInner.FieldNumber = 4 AND nU32 = TO_UDINT(E_SparkplugDataType.Float),
	sTestName  := 'T32 WriteFloatMetric datatype',
	nPass := nPass, nFail := nFail, sFirstFail := sFirstFail);

fbRInner.Next(); fbRInner.ReadFloat(fValue => fVal);
F_Assert(
	bCondition := fbRInner.FieldNumber = 12 AND fVal = 2.5,
	sTestName  := 'T33 WriteFloatMetric float_value (f12)',
	nPass := nPass, nFail := nFail, sFirstFail := sFirstFail);

// ── T34–T35: WriteDoubleMetric (double_value → proto field 13) ──────────────
fbPayload.Init(ADR(aBuf), SIZEOF(aBuf));
fbPayload.WriteHeader(nTestTs, 0);
fbPayload.WriteDoubleMetric('Pressure', 4, E_SparkplugDataType.Double, 0.125);

fbR.Init(fbPayload.Buffer, fbPayload.Length);
fbR.Next(); fbR.Skip(); fbR.Next(); fbR.Skip();
fbR.Next(); fbR.ReadBytes(pData => pMetric, nLen => nMetricLen);

fbRInner.Init(pMetric, nMetricLen);
fbRInner.Next(); fbRInner.Skip();
fbRInner.Next(); fbRInner.Skip();
fbRInner.Next(); fbRInner.ReadUInt32(nValue => nU32);
F_Assert(
	bCondition := fbRInner.FieldNumber = 4 AND nU32 = TO_UDINT(E_SparkplugDataType.Double),
	sTestName  := 'T34 WriteDoubleMetric datatype',
	nPass := nPass, nFail := nFail, sFirstFail := sFirstFail);

fbRInner.Next(); fbRInner.ReadDouble(fValue => dVal);
F_Assert(
	bCondition := fbRInner.FieldNumber = 13 AND dVal = 0.125,
	sTestName  := 'T35 WriteDoubleMetric double_value (f13)',
	nPass := nPass, nFail := nFail, sFirstFail := sFirstFail);

// ── T36–T37: WriteStringMetric (string_value → proto field 15) ──────────────
fbPayload.Init(ADR(aBuf), SIZEOF(aBuf));
fbPayload.WriteHeader(nTestTs, 0);
fbPayload.WriteStringMetric('Tag', 5, E_SparkplugDataType.String_, 'online');

fbR.Init(fbPayload.Buffer, fbPayload.Length);
fbR.Next(); fbR.Skip(); fbR.Next(); fbR.Skip();
fbR.Next(); fbR.ReadBytes(pData => pMetric, nLen => nMetricLen);

fbRInner.Init(pMetric, nMetricLen);
fbRInner.Next(); fbRInner.Skip();
fbRInner.Next(); fbRInner.Skip();
fbRInner.Next(); fbRInner.ReadUInt32(nValue => nU32);
F_Assert(
	bCondition := fbRInner.FieldNumber = 4 AND nU32 = TO_UDINT(E_SparkplugDataType.String_),
	sTestName  := 'T36 WriteStringMetric datatype',
	nPass := nPass, nFail := nFail, sFirstFail := sFirstFail);

fbRInner.Next(); fbRInner.ReadString(sValue => sVal);
F_Assert(
	bCondition := fbRInner.FieldNumber = 15 AND sVal = 'online',
	sTestName  := 'T37 WriteStringMetric string_value (f15)',
	nPass := nPass, nFail := nFail, sFirstFail := sFirstFail);


// ════════════════════════════════════════════════════════════════════════════
// Done
// ════════════════════════════════════════════════════════════════════════════
bAllPassed := (nFail = 0);
bRan       := TRUE;

END_PROGRAM
